// TwinCAT 3 PLC project popa_supervisor
// ProgramVersion: 3.1.4024.0
// libraries:
//   Tc2_ModbusSrv, * (Beckhoff Automation GmbH)
//   Tc2_Standard, * (Beckhoff Automation GmbH)
//   Tc2_System, * (Beckhoff Automation GmbH)
//   Tc2_Utilities, * (Beckhoff Automation GmbH)
//   Tc3_Module, * (Beckhoff Automation GmbH)
//   Tc2_OpcUa,3.3.2.0,Beckhoff Automation GmbH
// project tree:
//   DUTs/ U_Convert.TcDUT
//   GVLs/ heartbeat.TcGVL, opc.TcGVL
//   / PlcTask.TcTTO
//   POUs/ alarm_manager.TcPOU, eap_mapping.TcPOU, example_loop_control.TcPOU, faults.TcPOU, heartbeat_routine.TcPOU, interlocks.TcPOU, io_mapping.TcPOU, communications.TcPOU, general.TcPOU, modbus_mapping.TcPOU, motor_starter_control_st.TcPOU, motor_vfd_control_st.TcPOU, opc_control.TcPOU (not stored), opc_mapping.TcPOU, state_transition.TcPOU, valve_analog_control_st.TcPOU, valve_digital_control_st.TcPOU
//   POUs/Function Blocks/ int_arr_to_real.TcPOU, int_arr_to_real_1.TcPOU, modbus_analog_read.TcPOU, schneider_modbus_read.TcPOU, alarm.TcPOU, analog_scaling.TcPOU, date_time.TcPOU, motor_starter.TcPOU, motor_vfd.TcPOU, valve_analog.TcPOU, valve_digital.TcPOU
// real-time tasks:
//   TASK PlcTask: cycle T#10ms, priority 20, ADS port 350
// I/O:
//   DEVICE Device 1 (EtherCAT Automation Protocol), AmsNetId 10.60.1.100.2.1
//     Sup_Barge (Publisher)
//     Sup_Prexfer (Publisher)
//     Sup_ED (Publisher)
//     Sup_ProdXfer (Publisher)
//     Sup_Acid (Publisher)
//     Barge_Sup (Subscriber)
//     Prexfer_Sup (Subscriber)
//     ED_Sup (Subscriber)
//     ProdXfer_Sup (Subscriber)
//     Acid_Sup (Subscriber)
//   DEVICE Device 5 (EtherCAT), AmsNetId 10.60.1.100.6.1
//     Term 11 (EK1100) [EK1100 EtherCAT Coupler (2A E-Bus)]
//       Term 12 (EL2911) [EL2911, Potential supply terminal (10 A) with 4 Ch. Safety Inputs, TwinSAFE]
//         modules: Module 2 (FSOUT), Module 3 (DEVICEIO), Module 4 (FSLOGIC)
//       Term 3 (EL9011) [EL9011 End Terminal]
// variable links:
//   popa_supervisor Instance <-> Device 1 (EtherCAT Automation Protocol)/Acid_Sup (Subscriber)
//     PlcTask Inputs/eap_mapping.acid_critical_alarm <-> acid_critical_alarm/Inputs/VarData
//     PlcTask Inputs/eap_mapping.acid_error_alarm <-> acid_error_alarm/Inputs/VarData
//     PlcTask Inputs/eap_mapping.acid_warning_alarm <-> acid_warning_alarm/Inputs/VarData
//   popa_supervisor Instance <-> Device 1 (EtherCAT Automation Protocol)/Barge_Sup (Subscriber)
//     PlcTask Inputs/eap_mapping.barge_critical_alarm <-> barge_critical_alarm/Inputs/VarData
//     PlcTask Inputs/eap_mapping.barge_error_alarm <-> barge_error_alarm/Inputs/VarData
//     PlcTask Inputs/eap_mapping.barge_warning_alarm <-> barge_warning_alarm/Inputs/+
//   popa_supervisor Instance <-> Device 1 (EtherCAT Automation Protocol)/ED_Sup (Subscriber)
//     PlcTask Inputs/eap_mapping.ed_critical_alarm <-> ed_critical_alarm/Inputs/VarData
//     PlcTask Inputs/eap_mapping.ed_error_alarm <-> ed_error_alarm/Inputs/VarData
//     PlcTask Inputs/eap_mapping.ed_warning_alarm <-> ed_warning_alarm/Inputs/VarData
//   popa_supervisor Instance <-> Device 1 (EtherCAT Automation Protocol)/Prexfer_Sup (Subscriber)
//     PlcTask Inputs/eap_mapping.prexfer_critical_alarm <-> prexfer_critical_alarm/Inputs/VarData
//     PlcTask Inputs/eap_mapping.prexfer_error_alarm <-> prexfer_error_alarm/Inputs/VarData
//     PlcTask Inputs/eap_mapping.prexfer_warning_alarm <-> prexfer_warning_alarm/Inputs/VarData
//   popa_supervisor Instance <-> Device 1 (EtherCAT Automation Protocol)/ProdXfer_Sup (Subscriber)
//     PlcTask Inputs/eap_mapping.prodxfer_critical_alarm <-> prodxfer_critical_alarm/Inputs/VarData
//     PlcTask Inputs/eap_mapping.prodxfer_error_alarm <-> prodxfer_error_alarm/Inputs/VarData
//     PlcTask Inputs/eap_mapping.prodxfer_warning_alarm <-> prodxfer_warning_alarm/Inputs/VarData
//   popa_supervisor Instance <-> Device 1 (EtherCAT Automation Protocol)/Sup_Acid (Publisher)
//     PlcTask Outputs/eap_mapping.sup_acid_critical_alarm <-> sup_acid_critical_active/Outputs/VarData
//     PlcTask Outputs/eap_mapping.sup_acid_error_alarm <-> sup_acid_error_active/Outputs/VarData
//     PlcTask Outputs/eap_mapping.sup_acid_warning_alarm <-> sup_acid_warning_active/Outputs/VarData
//   popa_supervisor Instance <-> Device 1 (EtherCAT Automation Protocol)/Sup_Barge (Publisher)
//     PlcTask Outputs/eap_mapping.sup_barge_critical_alarm <-> Sup_Barge_Critical_Active/Outputs/VarData
//     PlcTask Outputs/eap_mapping.sup_barge_error_alarm <-> Sup_Barge_Error_Active/Outputs/VarData
//     PlcTask Outputs/eap_mapping.sup_barge_warning_alarm <-> Sup_Barge_Warning_Active/Outputs/VarData
//   popa_supervisor Instance <-> Device 1 (EtherCAT Automation Protocol)/Sup_ED (Publisher)
//     PlcTask Outputs/eap_mapping.sup_ed_critical_alarm <-> sup_ed_critical_active/Outputs/VarData
//     PlcTask Outputs/eap_mapping.sup_ed_error_alarm <-> sup_ed_error_active/Outputs/VarData
//     PlcTask Outputs/eap_mapping.sup_ed_warning_alarm <-> sup_ed_warning_active/Outputs/VarData
//   popa_supervisor Instance <-> Device 1 (EtherCAT Automation Protocol)/Sup_Prexfer (Publisher)
//     PlcTask Outputs/eap_mapping.sup_prexfer_critical_alarm <-> sup_prexfer_critical_active/Outputs/VarData
//     PlcTask Outputs/eap_mapping.sup_prexfer_error_alarm <-> sup_prexfer_error_active/Outputs/VarData
//     PlcTask Outputs/eap_mapping.sup_prexfer_warning_alarm <-> sup_prexfer_warning_active/Outputs/VarData
//   popa_supervisor Instance <-> Device 1 (EtherCAT Automation Protocol)/Sup_ProdXfer (Publisher)
//     PlcTask Outputs/eap_mapping.sup_prodxfer_critical_alarm <-> sup_prodxfer_critical_active/Outputs/VarData
//     PlcTask Outputs/eap_mapping.sup_prodxfer_error_alarm <-> sup_prodxfer_error_active/Outputs/VarData
//     PlcTask Outputs/eap_mapping.sup_prodxfer_warning_alarm <-> sup_prodxfer_warning_active/Outputs/VarData
//   popa_supervisor Instance <-> Device 5 (EtherCAT)/Term 11 (EK1100)/Term 12 (EL2911)
//     PlcTask Outputs/general.safety_error_ack <-> StandardOutputs/Standard In Var 1
//     PlcTask Outputs/general.safety_reset <-> StandardOutputs/Standard In Var 2
//     PlcTask Outputs/general.safety_run <-> StandardOutputs/Standard In Var 4

CONFIGURATION popa_supervisor
    RESOURCE PLC ON TwinCAT3
        TASK PlcTask(INTERVAL := T#10ms, PRIORITY := 20);
        PROGRAM communications WITH PlcTask : communications;
        PROGRAM example_loop_control WITH PlcTask : example_loop_control;
        PROGRAM faults WITH PlcTask : faults;
        PROGRAM general WITH PlcTask : general;
        PROGRAM interlocks WITH PlcTask : interlocks;
        PROGRAM io_mapping WITH PlcTask : io_mapping;
        PROGRAM opc_control WITH PlcTask : opc_control;
        PROGRAM opc_mapping WITH PlcTask : opc_mapping;
        PROGRAM state_transition WITH PlcTask : state_transition;
        PROGRAM eap_mapping WITH PlcTask : eap_mapping;
        PROGRAM alarm_manager WITH PlcTask : alarm_manager;
        PROGRAM modbus_mapping WITH PlcTask : modbus_mapping;
        PROGRAM heartbeat_routine WITH PlcTask : heartbeat_routine;
    END_RESOURCE
END_CONFIGURATION

// ---- DUTs/U_Convert.TcDUT
TYPE U_Convert :
UNION
	arrUDP_Data: ARRAY [0 .. 3] OF BYTE; // Array must start with LSB  
    rReal : REAL;
END_UNION
END_TYPE

// ---- GVLs/heartbeat.TcGVL
{attribute 'qualified_only'}
VAR_GLOBAL
	//OPC Bridge Heartbeat -- Logic found in heartbeat routine
	{attribute 'OPC.UA.DA' :='1'}
	opc_bridge_heartbeat : INT;
END_VAR

// ---- GVLs/opc.TcGVL
{attribute 'qualified_only'}
{attribute ‘OPC.UA.DA’ := ‘1’}//{attribute 'global_init_slot' := '50500'}
VAR_GLOBAL PERSISTENT
	//These tags are created here because you cannot write directly to local scoped tags(cpt_3144) from outside the POU
	//They are created here then mapped to the local variables in the POU
	//All tags in this GVL MUST have the {attribute 'OPC.UA.DA' :='1'} string above them in order to be exposed to OPC
	//Tags that are ONLY being read from the HMI have their values set in the opc_mapping program
		
	
	//--- Heartbeat ------------------------------------------------------------------------------------------------
	{attribute 'OPC.UA.DA' :='1'}
	popa_supervisor_opc_bridge_heartbeat : BOOL;
	
	//--- Safety ---------------------------------------------------------------------------------------------------
	{attribute 'OPC.UA.DA' :='1'}
	popa_supervisor_safety_reset : BOOL;
	
	{attribute 'OPC.UA.DA' :='1'}
	popa_supervisor_estop_active : BOOL;
	
	{attribute 'OPC.UA.DA' :='1'}
	popa_supervisor_barge_safety_triggered : BOOL;

	{attribute 'OPC.UA.DA' :='1'}
	popa_supervisor_ptt_safety_triggered : BOOL;

	{attribute 'OPC.UA.DA' :='1'}
	popa_supervisor_ed_safety_triggered : BOOL;

	{attribute 'OPC.UA.DA' :='1'}
	popa_supervisor_pdt_safety_triggered : BOOL;

	{attribute 'OPC.UA.DA' :='1'}
	popa_supervisor_acid_safety_triggered : BOOL;


	//--- Macoma Power Meters --------------------------------------------------------------------------------------

	{attribute 'OPC.UA.DA' :='1'}
	popa_supervisor_kt_3710_line_to_neutral_voltage_scaled_value : REAL;
	{attribute 'OPC.UA.DA' :='1'}
	popa_supervisor_kt_3710_line_to_line_voltage_scaled_value : REAL;
	{attribute 'OPC.UA.DA' :='1'}
	popa_supervisor_kt_3710_avg_line_current_scaled_value : REAL;
	{attribute 'OPC.UA.DA' :='1'}
	popa_supervisor_kt_3710_total_active_power_scaled_value : REAL;
	{attribute 'OPC.UA.DA' :='1'}
	popa_supervisor_kt_3710_total_reactive_power_scaled_value : REAL;
	{attribute 'OPC.UA.DA' :='1'}
	popa_supervisor_kt_3710_total_apparent_power_scaled_value : REAL;
	{attribute 'OPC.UA.DA' :='1'}
	popa_supervisor_kt_3710_total_power_factor_scaled_value : REAL;
	{attribute 'OPC.UA.DA' :='1'}
	popa_supervisor_kt_3710_system_frequency_scaled_value : REAL;
	
	{attribute 'OPC.UA.DA' :='1'}
	popa_supervisor_kt_3715_line_to_neutral_voltage_scaled_value : REAL;
	{attribute 'OPC.UA.DA' :='1'}
	popa_supervisor_kt_3715_line_to_line_voltage_scaled_value : REAL;
	{attribute 'OPC.UA.DA' :='1'}
	popa_supervisor_kt_3715_avg_line_current_scaled_value : REAL;
	{attribute 'OPC.UA.DA' :='1'}
	popa_supervisor_kt_3715_total_active_power_scaled_value : REAL;
	{attribute 'OPC.UA.DA' :='1'}
	popa_supervisor_kt_3715_total_reactive_power_scaled_value : REAL;
	{attribute 'OPC.UA.DA' :='1'}
	popa_supervisor_kt_3715_total_apparent_power_scaled_value : REAL;
	{attribute 'OPC.UA.DA' :='1'}
	popa_supervisor_kt_3715_total_power_factor_scaled_value : REAL;
	{attribute 'OPC.UA.DA' :='1'}
	popa_supervisor_kt_3715_system_frequency_scaled_value : REAL;
	
	{attribute 'OPC.UA.DA' :='1'}
	popa_supervisor_kt_2710_line_to_neutral_voltage_scaled_value : REAL;
	{attribute 'OPC.UA.DA' :='1'}
	popa_supervisor_kt_2710_line_to_line_voltage_scaled_value : REAL;
	{attribute 'OPC.UA.DA' :='1'}
	popa_supervisor_kt_2710_avg_line_current_scaled_value : REAL;
	{attribute 'OPC.UA.DA' :='1'}
	popa_supervisor_kt_2710_total_active_power_scaled_value : REAL;
	{attribute 'OPC.UA.DA' :='1'}
	popa_supervisor_kt_2710_total_reactive_power_scaled_value : REAL;
	{attribute 'OPC.UA.DA' :='1'}
	popa_supervisor_kt_2710_total_apparent_power_scaled_value : REAL;
	{attribute 'OPC.UA.DA' :='1'}
	popa_supervisor_kt_2710_total_power_factor_scaled_value : REAL;
	{attribute 'OPC.UA.DA' :='1'}
	popa_supervisor_kt_2710_system_frequency_scaled_value : REAL;
	
	{attribute 'OPC.UA.DA' :='1'}
	popa_supervisor_kt_2715_line_to_neutral_voltage_scaled_value : REAL;
	{attribute 'OPC.UA.DA' :='1'}
	popa_supervisor_kt_2715_line_to_line_voltage_scaled_value : REAL;
	{attribute 'OPC.UA.DA' :='1'}
	popa_supervisor_kt_2715_avg_line_current_scaled_value : REAL;
	{attribute 'OPC.UA.DA' :='1'}
	popa_supervisor_kt_2715_total_active_power_scaled_value : REAL;
	{attribute 'OPC.UA.DA' :='1'}
	popa_supervisor_kt_2715_total_reactive_power_scaled_value : REAL;
	{attribute 'OPC.UA.DA' :='1'}
	popa_supervisor_kt_2715_total_apparent_power_scaled_value : REAL;
	{attribute 'OPC.UA.DA' :='1'}
	popa_supervisor_kt_2715_total_power_factor_scaled_value : REAL;
	{attribute 'OPC.UA.DA' :='1'}
	popa_supervisor_kt_2715_system_frequency_scaled_value : REAL;
	
	
	{attribute 'OPC.UA.DA' :='1'}
	popa_supervisor_kt_2720_line_to_neutral_voltage_scaled_value : REAL;
	{attribute 'OPC.UA.DA' :='1'}
	popa_supervisor_kt_2720_line_to_line_voltage_scaled_value : REAL;
	{attribute 'OPC.UA.DA' :='1'}
	popa_supervisor_kt_2720_avg_line_current_scaled_value : REAL;
	{attribute 'OPC.UA.DA' :='1'}
	popa_supervisor_kt_2720_total_active_power_scaled_value : REAL;
	{attribute 'OPC.UA.DA' :='1'}
	popa_supervisor_kt_2720_total_reactive_power_scaled_value : REAL;
	{attribute 'OPC.UA.DA' :='1'}
	popa_supervisor_kt_2720_total_apparent_power_scaled_value : REAL;
	{attribute 'OPC.UA.DA' :='1'}
	popa_supervisor_kt_2720_total_power_factor_scaled_value : REAL;
	{attribute 'OPC.UA.DA' :='1'}
	popa_supervisor_kt_2720_system_frequency_scaled_value : REAL;
	
	{attribute 'OPC.UA.DA' :='1'}
	popa_supervisor_kt_2725_line_to_neutral_voltage_scaled_value : REAL;
	{attribute 'OPC.UA.DA' :='1'}
	popa_supervisor_kt_2725_line_to_line_voltage_scaled_value : REAL;
	{attribute 'OPC.UA.DA' :='1'}
	popa_supervisor_kt_2725_avg_line_current_scaled_value : REAL;
	{attribute 'OPC.UA.DA' :='1'}
	popa_supervisor_kt_2725_total_active_power_scaled_value : REAL;
	{attribute 'OPC.UA.DA' :='1'}
	popa_supervisor_kt_2725_total_reactive_power_scaled_value : REAL;
	{attribute 'OPC.UA.DA' :='1'}
	popa_supervisor_kt_2725_total_apparent_power_scaled_value : REAL;
	{attribute 'OPC.UA.DA' :='1'}
	popa_supervisor_kt_2725_total_power_factor_scaled_value : REAL;
	{attribute 'OPC.UA.DA' :='1'}
	popa_supervisor_kt_2725_system_frequency_scaled_value : REAL;
	
	{attribute 'OPC.UA.DA' :='1'}
	popa_supervisor_kt_2730_line_to_neutral_voltage_scaled_value : REAL;
	{attribute 'OPC.UA.DA' :='1'}
	popa_supervisor_kt_2730_line_to_line_voltage_scaled_value : REAL;
	{attribute 'OPC.UA.DA' :='1'}
	popa_supervisor_kt_2730_avg_line_current_scaled_value : REAL;
	{attribute 'OPC.UA.DA' :='1'}
	popa_supervisor_kt_2730_total_active_power_scaled_value : REAL;
	{attribute 'OPC.UA.DA' :='1'}
	popa_supervisor_kt_2730_total_reactive_power_scaled_value : REAL;
	{attribute 'OPC.UA.DA' :='1'}
	popa_supervisor_kt_2730_total_apparent_power_scaled_value : REAL;
	{attribute 'OPC.UA.DA' :='1'}
	popa_supervisor_kt_2730_total_power_factor_scaled_value : REAL;
	{attribute 'OPC.UA.DA' :='1'}
	popa_supervisor_kt_2730_system_frequency_scaled_value : REAL;
	
	{attribute 'OPC.UA.DA' :='1'}
	popa_supervisor_kt_3720_line_to_neutral_voltage_scaled_value : REAL;
	{attribute 'OPC.UA.DA' :='1'}
	popa_supervisor_kt_3720_line_to_line_voltage_scaled_value : REAL;
	{attribute 'OPC.UA.DA' :='1'}
	popa_supervisor_kt_3720_avg_line_current_scaled_value : REAL;
	{attribute 'OPC.UA.DA' :='1'}
	popa_supervisor_kt_3720_total_active_power_scaled_value : REAL;
	{attribute 'OPC.UA.DA' :='1'}
	popa_supervisor_kt_3720_total_reactive_power_scaled_value : REAL;
	{attribute 'OPC.UA.DA' :='1'}
	popa_supervisor_kt_3720_total_apparent_power_scaled_value : REAL;
	{attribute 'OPC.UA.DA' :='1'}
	popa_supervisor_kt_3720_total_power_factor_scaled_value : REAL;
	{attribute 'OPC.UA.DA' :='1'}
	popa_supervisor_kt_3720_system_frequency_scaled_value : REAL;
	
	{attribute 'OPC.UA.DA' :='1'}
	popa_supervisor_kt_1720_line_to_neutral_voltage_scaled_value : REAL;
	{attribute 'OPC.UA.DA' :='1'}
	popa_supervisor_kt_1720_line_to_line_voltage_scaled_value : REAL;
	{attribute 'OPC.UA.DA' :='1'}
	popa_supervisor_kt_1720_avg_line_current_scaled_value : REAL;
	{attribute 'OPC.UA.DA' :='1'}
	popa_supervisor_kt_1720_total_active_power_scaled_value : REAL;
	{attribute 'OPC.UA.DA' :='1'}
	popa_supervisor_kt_1720_total_reactive_power_scaled_value : REAL;
	{attribute 'OPC.UA.DA' :='1'}
	popa_supervisor_kt_1720_total_apparent_power_scaled_value : REAL;
	{attribute 'OPC.UA.DA' :='1'}
	popa_supervisor_kt_1720_total_power_factor_scaled_value : REAL;
	{attribute 'OPC.UA.DA' :='1'}
	popa_supervisor_kt_1720_system_frequency_scaled_value : REAL;
	
	{attribute 'OPC.UA.DA' :='1'}
	popa_supervisor_kt_4710_line_to_neutral_voltage_scaled_value : REAL;
	{attribute 'OPC.UA.DA' :='1'}
	popa_supervisor_kt_4710_line_to_line_voltage_scaled_value : REAL;
	{attribute 'OPC.UA.DA' :='1'}
	popa_supervisor_kt_4710_avg_line_current_scaled_value : REAL;
	{attribute 'OPC.UA.DA' :='1'}
	popa_supervisor_kt_4710_total_active_power_scaled_value : REAL;
	{attribute 'OPC.UA.DA' :='1'}
	popa_supervisor_kt_4710_total_reactive_power_scaled_value : REAL;
	{attribute 'OPC.UA.DA' :='1'}
	popa_supervisor_kt_4710_total_apparent_power_scaled_value : REAL;
	{attribute 'OPC.UA.DA' :='1'}
	popa_supervisor_kt_4710_total_power_factor_scaled_value : REAL;
	{attribute 'OPC.UA.DA' :='1'}
	popa_supervisor_kt_4710_system_frequency_scaled_value : REAL;
	
	{attribute 'OPC.UA.DA' :='1'}
	popa_supervisor_kt_1725_line_to_neutral_voltage_scaled_value : REAL;
	{attribute 'OPC.UA.DA' :='1'}
	popa_supervisor_kt_1725_line_to_line_voltage_scaled_value : REAL;
	{attribute 'OPC.UA.DA' :='1'}
	popa_supervisor_kt_1725_avg_line_current_scaled_value : REAL;
	{attribute 'OPC.UA.DA' :='1'}
	popa_supervisor_kt_1725_total_active_power_scaled_value : REAL;
	{attribute 'OPC.UA.DA' :='1'}
	popa_supervisor_kt_1725_total_reactive_power_scaled_value : REAL;
	{attribute 'OPC.UA.DA' :='1'}
	popa_supervisor_kt_1725_total_apparent_power_scaled_value : REAL;
	{attribute 'OPC.UA.DA' :='1'}
	popa_supervisor_kt_1725_total_power_factor_scaled_value : REAL;
	{attribute 'OPC.UA.DA' :='1'}
	popa_supervisor_kt_1725_system_frequency_scaled_value : REAL;
	
	{attribute 'OPC.UA.DA' :='1'}
	popa_supervisor_kt_1715_line_to_neutral_voltage_scaled_value : REAL;
	{attribute 'OPC.UA.DA' :='1'}
	popa_supervisor_kt_1715_line_to_line_voltage_scaled_value : REAL;
	{attribute 'OPC.UA.DA' :='1'}
	popa_supervisor_kt_1715_avg_line_current_scaled_value : REAL;
	{attribute 'OPC.UA.DA' :='1'}
	popa_supervisor_kt_1715_total_active_power_scaled_value : REAL;
	{attribute 'OPC.UA.DA' :='1'}
	popa_supervisor_kt_1715_total_reactive_power_scaled_value : REAL;
	{attribute 'OPC.UA.DA' :='1'}
	popa_supervisor_kt_1715_total_apparent_power_scaled_value : REAL;
	{attribute 'OPC.UA.DA' :='1'}
	popa_supervisor_kt_1715_total_power_factor_scaled_value : REAL;
	{attribute 'OPC.UA.DA' :='1'}
	popa_supervisor_kt_1715_system_frequency_scaled_value : REAL;
	{attribute 'OPC.UA.DA' :='1'}
	popa_supervisor_kt_1715_ground_current_scaled_value : REAL;
	{attribute 'OPC.UA.DA' :='1'}
	popa_supervisor_kt_1715_current_capacity_scaled_value : REAL;
	{attribute 'OPC.UA.DA' :='1'}
	popa_supervisor_kt_1715_power_factor_leading_scaled_value : REAL;
	{attribute 'OPC.UA.DA' :='1'}
	popa_supervisor_kt_1715_power_factor_lagging_scaled_value : REAL;
	
	{attribute 'OPC.UA.DA' :='1'}
	popa_supervisor_kt_1710_line_to_neutral_voltage_scaled_value : REAL;
	{attribute 'OPC.UA.DA' :='1'}
	popa_supervisor_kt_1710_line_to_line_voltage_scaled_value : REAL;
	{attribute 'OPC.UA.DA' :='1'}
	popa_supervisor_kt_1710_avg_line_current_scaled_value : REAL;
	{attribute 'OPC.UA.DA' :='1'}
	popa_supervisor_kt_1710_total_active_power_scaled_value : REAL;
	{attribute 'OPC.UA.DA' :='1'}
	popa_supervisor_kt_1710_total_reactive_power_scaled_value : REAL;
	{attribute 'OPC.UA.DA' :='1'}
	popa_supervisor_kt_1710_total_apparent_power_scaled_value : REAL;
	{attribute 'OPC.UA.DA' :='1'}
	popa_supervisor_kt_1710_total_power_factor_scaled_value : REAL;
	{attribute 'OPC.UA.DA' :='1'}
	popa_supervisor_kt_1710_system_frequency_scaled_value : REAL;
	{attribute 'OPC.UA.DA' :='1'}
	popa_supervisor_kt_1710_ground_current_scaled_value : REAL;
	{attribute 'OPC.UA.DA' :='1'}
	popa_supervisor_kt_1710_current_capacity_scaled_value : REAL;
	{attribute 'OPC.UA.DA' :='1'}
	popa_supervisor_kt_1710_power_factor_leading_scaled_value : REAL;
	{attribute 'OPC.UA.DA' :='1'}
	popa_supervisor_kt_1710_power_factor_lagging_scaled_value : REAL;

END_VAR

// ---- POUs/communications.TcPOU
PROGRAM communications
VAR PERSISTENT
END_VAR

END_PROGRAM

// ---- POUs/example_loop_control.TcPOU
PROGRAM example_loop_control
VAR

END_VAR

// NETWORK 1

END_PROGRAM

// ---- POUs/faults.TcPOU
PROGRAM faults
VAR PERSISTENT
	// Example analog alarm low low
	cpt_3144_low_low: Alarm;
	// Example analog alarm low
	cpt_3144_low: Alarm;
	// Example analog alarm high
	cpt_3144_high: Alarm;
	// Example analog alarm high high
	cpt_3144_high_high: Alarm;
END_VAR

(*//Instantiate the alarm block, and map the inputs from the OPC GVL
cpt_3144_low_low();
cpt_3144_low_low.alm_ack:=opc.popa_0081_alarm_ack;
cpt_3144_low_low.reset:=opc.popa_0081_alarm_reset;
cpt_3144_low_low.priority:=opc.popa_0081_cpt_3144_low_low_priority;
cpt_3144_low_low.delay_setpoint:=opc.popa_0081_cpt_3144_low_low_delay_setpoint;
cpt_3144_low_low.enable:=opc.popa_0081_cpt_3144_low_low_enable;

//Place your alarm trigger logic here.  
IF io_mapping.cpt_3144.scaled_value<opc.popa_0081_cpt_3144_low_low_setpoint THEN
	cpt_3144_low_low.trigger:=TRUE;
	ELSE
		cpt_3144_low_low.trigger:=FALSE;
	END_IF	
	
//Instantiate the alarm block, and map the inputs from the OPC GVL
cpt_3144_low();
cpt_3144_low.alm_ack:=opc.popa_0081_alarm_ack;
cpt_3144_low.reset:=opc.popa_0081_alarm_reset;
cpt_3144_low.priority:=opc.popa_0081_cpt_3144_low_priority;
cpt_3144_low.delay_setpoint:=opc.popa_0081_cpt_3144_low_delay_setpoint;
cpt_3144_low.enable:=opc.popa_0081_cpt_3144_low_enable;

//Place your alarm trigger logic here.  
IF io_mapping.cpt_3144.scaled_value<opc.popa_0081_cpt_3144_low_setpoint THEN
	cpt_3144_low.trigger:=TRUE;
	ELSE
		cpt_3144_low.trigger:=FALSE;
	END_IF
	
//Instantiate the alarm block, and map the inputs from the OPC GVL
cpt_3144_high();
cpt_3144_high.alm_ack:=opc.popa_0081_alarm_ack;
cpt_3144_high.reset:=opc.popa_0081_alarm_reset;
cpt_3144_high.priority:=opc.popa_0081_cpt_3144_high_priority;
cpt_3144_high.delay_setpoint:=opc.popa_0081_cpt_3144_high_delay_setpoint;
cpt_3144_high.enable:=opc.popa_0081_cpt_3144_high_enable;

//Place your alarm trigger logic here.  
IF io_mapping.cpt_3144.scaled_value<opc.popa_0081_cpt_3144_high_setpoint THEN
	cpt_3144_high.trigger:=TRUE;
	ELSE
		cpt_3144_high.trigger:=FALSE;
	END_IF
	
//Instantiate the alarm block, and map the inputs from the OPC GVL
cpt_3144_high_high();
cpt_3144_high_high.alm_ack:=opc.popa_0081_alarm_ack;
cpt_3144_high_high.reset:=opc.popa_0081_alarm_reset;
cpt_3144_high_high.priority:=opc.popa_0081_cpt_3144_high_high_priority;
cpt_3144_high_high.delay_setpoint:=opc.popa_0081_cpt_3144_high_high_delay_setpoint;
cpt_3144_high_high.enable:=opc.popa_0081_cpt_3144_high_high_enable;

//Place your alarm trigger logic here.  
IF io_mapping.cpt_3144.scaled_value<opc.popa_0081_cpt_3144_high_high_setpoint THEN
	cpt_3144_high_high.trigger:=TRUE;
	ELSE
		cpt_3144_high_high.trigger:=FALSE;
	END_IF
	*)

END_PROGRAM

// ---- POUs/Function Blocks/alarm.TcPOU
FUNCTION_BLOCK alarm
VAR_INPUT
	//Input that triggers the alarm condition
	trigger : BOOL;
	//Alarm Acknowledge bit, Clears low priority alarms
	alm_ack : BOOL;
	//Alarm Reset, clears high priority alarms
	reset : BOOL;
	//Alarm Priority, 1=Warning, 2=Error, 3=Critical
	priority : INT;
	//Alarm Delay Setpoint in Seconds
	delay_setpoint : INT;
	//Alarm Enable
	enable : BOOL;
END_VAR
VAR_OUTPUT
	//Alarm is triggered
	active : BOOL;
END_VAR
VAR
	//Delay Timer Tags
	delay_ton : TON;
	delay_ton_pt : TIME;
	delay_ton_et : TIME;
	//Delay setpoint converted to Milliseconds
	delay_ms : REAL;
	//Cutoff for needing to reset vs ack an alarm.  At or above this value requires reset.  
	reset_priority : REAL :=3;
END_VAR

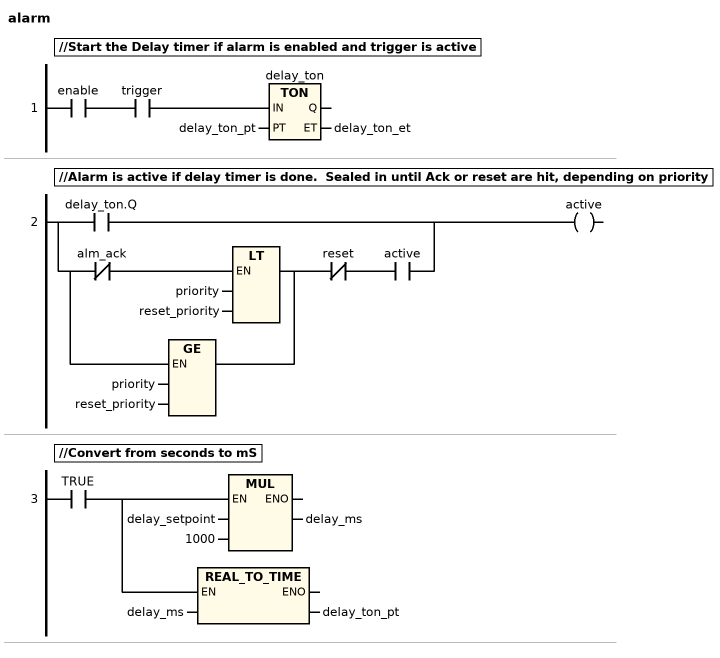
// NETWORK 1
// label: //Start the Delay timer if alarm is enabled and trigger is active
delay_ton(IN := enable AND trigger, PT := delay_ton_pt, ET => delay_ton_et); // TON

// NETWORK 2
// label: //Alarm is active if delay timer is done.  Sealed in until Ack or reset are hit, depending on priority
active := delay_ton.Q OR (NOT alm_ack AND priority < reset_priority OR priority >= reset_priority) AND NOT reset AND active;

// NETWORK 3
// label: //Convert from seconds to mS
delay_ms := delay_setpoint * 1000;
delay_ton_pt := REAL_TO_TIME(delay_ms);

END_FUNCTION_BLOCK

// ---- POUs/general.TcPOU
PROGRAM general
VAR PERSISTENT
	//System date time function block
	system_date_time : date_time;
	//Daily reset bit, used throughout the program for any resets
	daily_reset : BOOL;
	//Alarm Acknoweldge unlatch timer
	alarm_ack_ton : ton;
	//Alarm Reset unlatch timer
	alarm_reset_ton : ton;
	//Alarm Ack and reset unlatch timer setpoint
	alarm_ack_unlatch_sp : TIME :=T#3S;
	
	safety_reset_ton : TON;
	
	safety_reset AT %Q*  : BOOL;
	safety_error_ack AT %Q* : BOOL;
	safety_run AT %Q*  : BOOL;
	
END_VAR

VAR
	
	safety_reset_ons: R_TRIG;
END_VAR
VAR // added by the converter: edge detectors and wires of the graphical bodies
    _w1 : BOOL;
END_VAR

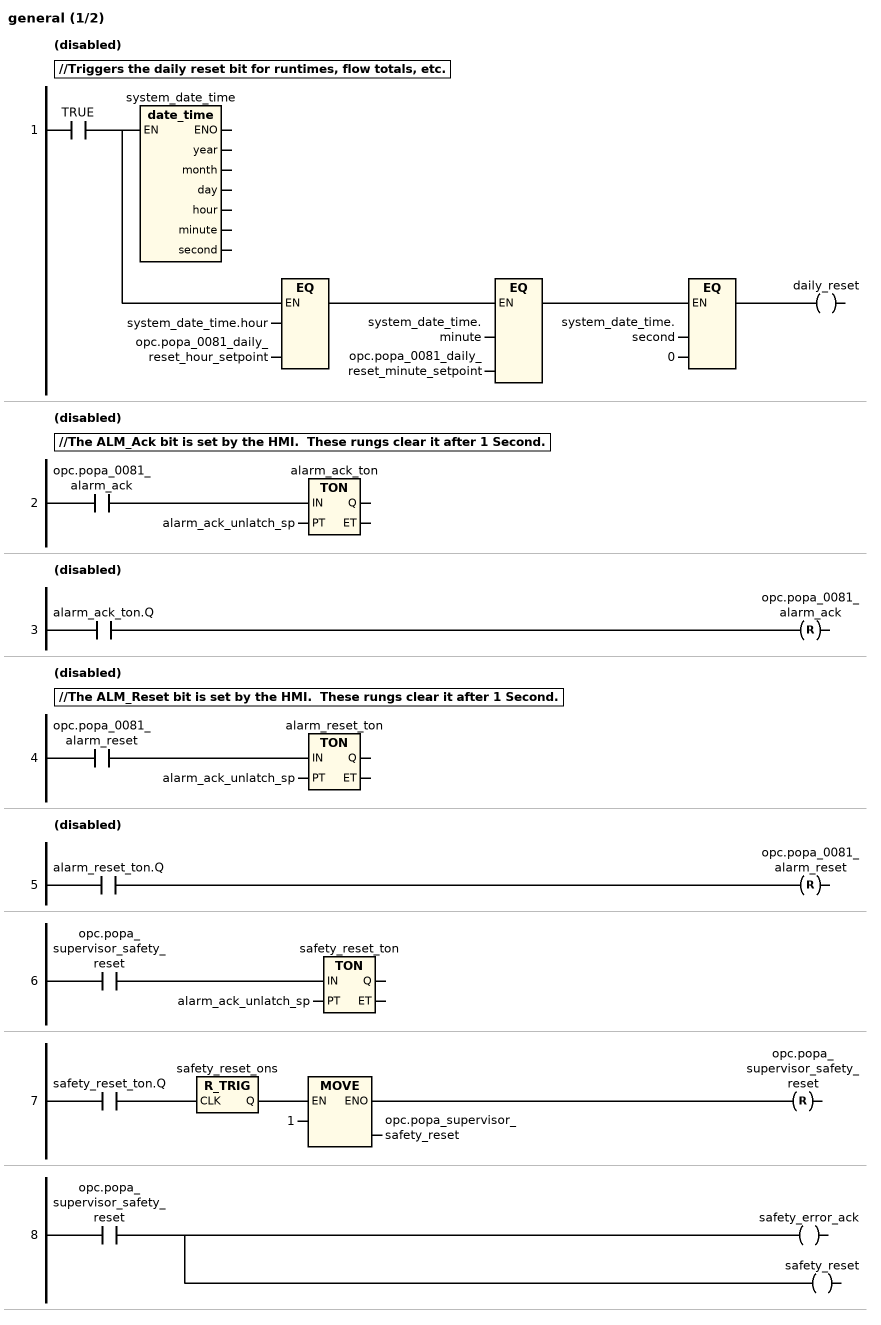
// NETWORK 1 (disabled)
// label: //Triggers the daily reset bit for runtimes, flow totals, etc.
// system_date_time(); // date_time
// daily_reset := system_date_time.hour = opc.popa_0081_daily_reset_hour_setpoint AND system_date_time.minute = opc.popa_0081_daily_reset_minute_setpoint AND system_date_time.second = 0;

// NETWORK 2 (disabled)
// label: //The ALM_Ack bit is set by the HMI.  These rungs clear it after 1 Second.
// alarm_ack_ton(IN := opc.popa_0081_alarm_ack, PT := alarm_ack_unlatch_sp); // TON

// NETWORK 3 (disabled)
// opc.popa_0081_alarm_ack R= alarm_ack_ton.Q;

// NETWORK 4 (disabled)
// label: //The ALM_Reset bit is set by the HMI.  These rungs clear it after 1 Second.
// alarm_reset_ton(IN := opc.popa_0081_alarm_reset, PT := alarm_ack_unlatch_sp); // TON

// NETWORK 5 (disabled)
// opc.popa_0081_alarm_reset R= alarm_reset_ton.Q;

// NETWORK 6
safety_reset_ton(IN := opc.popa_supervisor_safety_reset, PT := alarm_ack_unlatch_sp); // TON

// NETWORK 7
safety_reset_ons(CLK := safety_reset_ton.Q); // R_TRIG
_w1 := safety_reset_ons.Q;
IF _w1 THEN opc.popa_supervisor_safety_reset := 1; END_IF
opc.popa_supervisor_safety_reset R= _w1;

// NETWORK 8
safety_error_ack := opc.popa_supervisor_safety_reset;
safety_reset := opc.popa_supervisor_safety_reset;

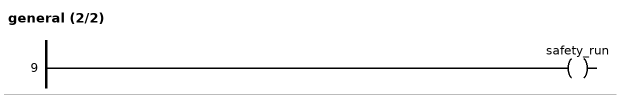
// NETWORK 9
safety_run := TRUE;

END_PROGRAM

// ---- POUs/Function Blocks/date_time.TcPOU
FUNCTION_BLOCK Date_Time
VAR_INPUT
END_VAR
VAR_OUTPUT
	Year : INT;
	Month : INT;
	Day : INT;
	Hour : INT;
	Minute : INT;
	Second : INT;
END_VAR
VAR
	fbGetSystemTime : GETSYSTEMTIME;    (*timestamp*)
    fileTime        : T_FILETIME;
    sDT: STRING(30);
END_VAR

//Get Timestamp from System
fbGetSystemTime(timeLoDW => fileTime.dwLowDateTime, timeHiDW => fileTime.dwHighDateTime);
//Convert from systemtime to string, this makes it easier to break out into Ints for Logic usage.
sDT := SYSTEMTIME_TO_STRING(FILETIME_TO_SYSTEMTIME(fileTime));
//Breakout string into individual Ints.
Year := STRING_TO_INT(LEFT(sDt, 4));
Month := STRING_TO_INT(MID(sDt, 2, 6));
Day := STRING_TO_INT(MID(sDt, 2, 9));
Hour := STRING_TO_INT(MID(sDt, 2, 12));
Minute := STRING_TO_INT(MID(sDt, 2, 15));
Second := STRING_TO_INT(MID(sDt, 2, 18));

END_FUNCTION_BLOCK

// ---- POUs/interlocks.TcPOU
PROGRAM interlocks
VAR PERSISTENT
END_VAR

// NETWORK 1

END_PROGRAM

// ---- POUs/io_mapping.TcPOU
PROGRAM io_mapping
VAR PERSISTENT
    //Example analog input function block
    cpt_3144 : analog_scaling;
	
	test_real AT %Q* : REAL;
	
	publisharray AT %Q* : ARRAY[0..9] OF REAL;
	
	sine_wave : REAL;
	
    //Example Analog input raw input, mapped to a physical input
    cpt_3144_raw_input AT %I* : INT;

END_VAR

(*//Instantiate Example analog input function block
cpt_3144();

//Map values from the OPC GVL so that they can be written to from outside POU(IE from HMI)
cpt_3144.eu_max:=opc.popa_0081_cpt_3144_eu_max;
cpt_3144.eu_min:=opc.popa_0081_cpt_3144_eu_min;
cpt_3144.filter_factor:=opc.popa_0081_cpt_3144_filter_factor;
cpt_3144.raw_max:=opc.popa_0081_cpt_3144_raw_max;
cpt_3144.raw_min:=opc.popa_0081_cpt_3144_raw_min;
//Map the analog scaling function block raw input to the physical raw input variable
cpt_3144.raw_input := cpt_3144_raw_input;

sine_wave:=sine_wave+0.001;
IF (sine_wave>(2*pi)) THEN
	sine_wave:=0;
END_IF
*)
publisharray[0]:=sine_wave;
publisharray[1]:=sine_wave/2;
publisharray[2]:=sine_wave*2;

END_PROGRAM

// ---- POUs/Function Blocks/analog_scaling.TcPOU
FUNCTION_BLOCK Analog_Scaling
VAR_INPUT
	//Raw Input value
	Raw_Input : REAL;
	//Raw Input Minimum Scaling Value
	Raw_Min : REAL;
	//Raw Input Maximum Scaling Value
	Raw_Max : REAL;
	//Engineering Units Minimum Scaling Value
	EU_Min : REAL;
	//Engineering Units Maximum Scaling Value
	EU_Max : REAL;
	//Averaging Filter Time Setpoint
	Filter_Factor : REAL;
END_VAR
VAR_OUTPUT
	//Scaled Value for Output
	Scaled_Value : REAL;
END_VAR
VAR
	//Scratchpad Value
	Normalized_Value : REAL;
	//Normalized/Scaled Value
	Scaled : REAL;
END_VAR

//Initialize Raw_Max and EU_Max to avoid Scaled_Value=Not a number
IF Raw_Max = 0 AND Raw_Min = 0 THEN
	Raw_Max:=1;
END_IF
IF EU_Max = 0 AND Raw_Min = 0 THEN
	EU_Max:=1;
END_IF

//Normalize the Analog Input
IF Raw_Input < Raw_Min THEN
		Normalized_Value := Raw_Min;
	ELSIF Raw_Input > Raw_Max THEN
		Normalized_Value := Raw_Max;
	ELSE
		Normalized_Value := (Raw_Input - Raw_Min) / (Raw_Max - Raw_Min);
	END_IF
	
//Scale the Output
Scaled := Normalized_Value * (EU_Max-EU_Min)+EU_Min;

//Low Pass Filter for the output.  Increase Filter to dampen reading
Scaled_Value := ((Scaled_Value * Filter_Factor) + Scaled) / (Filter_Factor +1);

END_FUNCTION_BLOCK

// ---- POUs/opc_mapping.TcPOU
PROGRAM opc_mapping
VAR
END_VAR

//This program maps values from the local variable to the OPC readable tag.
// --- Hearbeat ------------------------------------------------------------------------------------------------------------------------------------
opc.popa_supervisor_opc_bridge_heartbeat := NOT(heartbeat_routine.opc_heartbeat_error);

// --- Safety Logging ------------------------------------------------------------------------------------------------------------------------------
opc.popa_supervisor_barge_safety_triggered := eap_mapping.barge_critical_alarm;
opc.popa_supervisor_ptt_safety_triggered := eap_mapping.prexfer_critical_alarm;
opc.popa_supervisor_ed_safety_triggered := eap_mapping.ed_critical_alarm;
opc.popa_supervisor_pdt_safety_triggered := eap_mapping.prodxfer_critical_alarm;
opc.popa_supervisor_acid_safety_triggered := eap_mapping.acid_critical_alarm;

// --- Power Meter Data ----------------------------------------------------------------------------------------------------------------------------
opc.popa_supervisor_kt_3710_line_to_neutral_voltage_scaled_value := modbus_mapping.bped_main_power_meter_modbus_read.avg_line_to_neutral_voltage;

opc.popa_supervisor_kt_3710_line_to_line_voltage_scaled_value := modbus_mapping.bped_main_power_meter_modbus_read.avg_line_to_line_voltage;

opc.popa_supervisor_kt_3710_avg_line_current_scaled_value := modbus_mapping.bped_main_power_meter_modbus_read.system_avg_line_current;

opc.popa_supervisor_kt_3710_total_active_power_scaled_value := modbus_mapping.bped_main_power_meter_modbus_read.total_active_power;

opc.popa_supervisor_kt_3710_total_reactive_power_scaled_value := modbus_mapping.bped_main_power_meter_modbus_read.total_reactive_power;

opc.popa_supervisor_kt_3710_total_apparent_power_scaled_value := modbus_mapping.bped_main_power_meter_modbus_read.total_apparent_power;

opc.popa_supervisor_kt_3710_total_power_factor_scaled_value := modbus_mapping.bped_main_power_meter_modbus_read.total_power_factor;

opc.popa_supervisor_kt_3710_system_frequency_scaled_value := modbus_mapping.bped_main_power_meter_modbus_read.system_frequency;

opc.popa_supervisor_kt_3715_line_to_neutral_voltage_scaled_value := modbus_mapping.bped_stack_power_meter_modbus_read.avg_line_to_neutral_voltage;

opc.popa_supervisor_kt_3715_line_to_line_voltage_scaled_value := modbus_mapping.bped_stack_power_meter_modbus_read.avg_line_to_line_voltage;

opc.popa_supervisor_kt_3715_avg_line_current_scaled_value := modbus_mapping.bped_stack_power_meter_modbus_read.system_avg_line_current;

opc.popa_supervisor_kt_3715_total_active_power_scaled_value := modbus_mapping.bped_stack_power_meter_modbus_read.total_active_power;

opc.popa_supervisor_kt_3715_total_reactive_power_scaled_value := modbus_mapping.bped_stack_power_meter_modbus_read.total_reactive_power;

opc.popa_supervisor_kt_3715_total_apparent_power_scaled_value := modbus_mapping.bped_stack_power_meter_modbus_read.total_apparent_power;

opc.popa_supervisor_kt_3715_total_power_factor_scaled_value := modbus_mapping.bped_stack_power_meter_modbus_read.total_power_factor;

opc.popa_supervisor_kt_3715_system_frequency_scaled_value := modbus_mapping.bped_stack_power_meter_modbus_read.system_frequency;


opc.popa_supervisor_kt_2710_line_to_neutral_voltage_scaled_value := modbus_mapping.nf1_power_meter_modbus_read.avg_line_to_neutral_voltage;

opc.popa_supervisor_kt_2710_line_to_line_voltage_scaled_value := modbus_mapping.nf1_power_meter_modbus_read.avg_line_to_line_voltage;

opc.popa_supervisor_kt_2710_avg_line_current_scaled_value := modbus_mapping.nf1_power_meter_modbus_read.system_avg_line_current;

opc.popa_supervisor_kt_2710_total_active_power_scaled_value := modbus_mapping.nf1_power_meter_modbus_read.total_active_power;

opc.popa_supervisor_kt_2710_total_reactive_power_scaled_value := modbus_mapping.nf1_power_meter_modbus_read.total_reactive_power;

opc.popa_supervisor_kt_2710_total_apparent_power_scaled_value := modbus_mapping.nf1_power_meter_modbus_read.total_apparent_power;

opc.popa_supervisor_kt_2710_total_power_factor_scaled_value := modbus_mapping.nf1_power_meter_modbus_read.total_power_factor;

opc.popa_supervisor_kt_2710_system_frequency_scaled_value := modbus_mapping.nf1_power_meter_modbus_read.system_frequency;


opc.popa_supervisor_kt_2715_line_to_neutral_voltage_scaled_value := modbus_mapping.nf2_power_meter_modbus_read.avg_line_to_neutral_voltage;

opc.popa_supervisor_kt_2715_line_to_line_voltage_scaled_value := modbus_mapping.nf2_power_meter_modbus_read.avg_line_to_line_voltage;

opc.popa_supervisor_kt_2715_avg_line_current_scaled_value := modbus_mapping.nf2_power_meter_modbus_read.system_avg_line_current;

opc.popa_supervisor_kt_2715_total_active_power_scaled_value := modbus_mapping.nf2_power_meter_modbus_read.total_active_power;

opc.popa_supervisor_kt_2715_total_reactive_power_scaled_value := modbus_mapping.nf2_power_meter_modbus_read.total_reactive_power;

opc.popa_supervisor_kt_2715_total_apparent_power_scaled_value := modbus_mapping.nf2_power_meter_modbus_read.total_apparent_power;

opc.popa_supervisor_kt_2715_total_power_factor_scaled_value := modbus_mapping.nf2_power_meter_modbus_read.total_power_factor;

opc.popa_supervisor_kt_2715_system_frequency_scaled_value := modbus_mapping.nf2_power_meter_modbus_read.system_frequency;



opc.popa_supervisor_kt_2720_line_to_neutral_voltage_scaled_value := modbus_mapping.ro_power_meter_modbus_read.avg_line_to_neutral_voltage;

opc.popa_supervisor_kt_2720_line_to_line_voltage_scaled_value := modbus_mapping.ro_power_meter_modbus_read.avg_line_to_line_voltage;

opc.popa_supervisor_kt_2720_avg_line_current_scaled_value := modbus_mapping.ro_power_meter_modbus_read.system_avg_line_current;

opc.popa_supervisor_kt_2720_total_active_power_scaled_value := modbus_mapping.ro_power_meter_modbus_read.total_active_power;

opc.popa_supervisor_kt_2720_total_reactive_power_scaled_value := modbus_mapping.ro_power_meter_modbus_read.total_reactive_power;

opc.popa_supervisor_kt_2720_total_apparent_power_scaled_value := modbus_mapping.ro_power_meter_modbus_read.total_apparent_power;

opc.popa_supervisor_kt_2720_total_power_factor_scaled_value := modbus_mapping.ro_power_meter_modbus_read.total_power_factor;

opc.popa_supervisor_kt_2720_system_frequency_scaled_value := modbus_mapping.ro_power_meter_modbus_read.system_frequency;


opc.popa_supervisor_kt_2725_line_to_neutral_voltage_scaled_value := modbus_mapping.rocip_power_meter_modbus_read.avg_line_to_neutral_voltage;

opc.popa_supervisor_kt_2725_line_to_line_voltage_scaled_value := modbus_mapping.rocip_power_meter_modbus_read.avg_line_to_line_voltage;

opc.popa_supervisor_kt_2725_avg_line_current_scaled_value := modbus_mapping.rocip_power_meter_modbus_read.system_avg_line_current;

opc.popa_supervisor_kt_2725_total_active_power_scaled_value := modbus_mapping.rocip_power_meter_modbus_read.total_active_power;

opc.popa_supervisor_kt_2725_total_reactive_power_scaled_value := modbus_mapping.rocip_power_meter_modbus_read.total_reactive_power;

opc.popa_supervisor_kt_2725_total_apparent_power_scaled_value := modbus_mapping.rocip_power_meter_modbus_read.total_apparent_power;

opc.popa_supervisor_kt_2725_total_power_factor_scaled_value := modbus_mapping.rocip_power_meter_modbus_read.total_power_factor;

opc.popa_supervisor_kt_2725_system_frequency_scaled_value := modbus_mapping.rocip_power_meter_modbus_read.system_frequency;


opc.popa_supervisor_kt_2730_line_to_neutral_voltage_scaled_value := modbus_mapping.prexfer_power_meter_modbus_read.avg_line_to_neutral_voltage;

opc.popa_supervisor_kt_2730_line_to_line_voltage_scaled_value := modbus_mapping.prexfer_power_meter_modbus_read.avg_line_to_line_voltage;

opc.popa_supervisor_kt_2730_avg_line_current_scaled_value := modbus_mapping.prexfer_power_meter_modbus_read.system_avg_line_current;

opc.popa_supervisor_kt_2730_total_active_power_scaled_value := modbus_mapping.prexfer_power_meter_modbus_read.total_active_power;

opc.popa_supervisor_kt_2730_total_reactive_power_scaled_value := modbus_mapping.prexfer_power_meter_modbus_read.total_reactive_power;

opc.popa_supervisor_kt_2730_total_apparent_power_scaled_value := modbus_mapping.prexfer_power_meter_modbus_read.total_apparent_power;

opc.popa_supervisor_kt_2730_total_power_factor_scaled_value := modbus_mapping.prexfer_power_meter_modbus_read.total_power_factor;

opc.popa_supervisor_kt_2730_system_frequency_scaled_value := modbus_mapping.prexfer_power_meter_modbus_read.system_frequency;


opc.popa_supervisor_kt_3720_line_to_neutral_voltage_scaled_value := modbus_mapping.bop_power_meter_modbus_read.avg_line_to_neutral_voltage;

opc.popa_supervisor_kt_3720_line_to_line_voltage_scaled_value := modbus_mapping.bop_power_meter_modbus_read.avg_line_to_line_voltage;

opc.popa_supervisor_kt_3720_avg_line_current_scaled_value := modbus_mapping.bop_power_meter_modbus_read.system_avg_line_current;

opc.popa_supervisor_kt_3720_total_active_power_scaled_value := modbus_mapping.bop_power_meter_modbus_read.total_active_power;

opc.popa_supervisor_kt_3720_total_reactive_power_scaled_value := modbus_mapping.bop_power_meter_modbus_read.total_reactive_power;

opc.popa_supervisor_kt_3720_total_apparent_power_scaled_value := modbus_mapping.bop_power_meter_modbus_read.total_apparent_power;

opc.popa_supervisor_kt_3720_total_power_factor_scaled_value := modbus_mapping.bop_power_meter_modbus_read.total_power_factor;

opc.popa_supervisor_kt_3720_system_frequency_scaled_value := modbus_mapping.bop_power_meter_modbus_read.system_frequency;


opc.popa_supervisor_kt_1720_line_to_neutral_voltage_scaled_value := modbus_mapping.prodxfer_power_meter_modbus_read.avg_line_to_neutral_voltage;

opc.popa_supervisor_kt_1720_line_to_line_voltage_scaled_value := modbus_mapping.prodxfer_power_meter_modbus_read.avg_line_to_line_voltage;

opc.popa_supervisor_kt_1720_avg_line_current_scaled_value := modbus_mapping.prodxfer_power_meter_modbus_read.system_avg_line_current;

opc.popa_supervisor_kt_1720_total_active_power_scaled_value := modbus_mapping.prodxfer_power_meter_modbus_read.total_active_power;

opc.popa_supervisor_kt_1720_total_reactive_power_scaled_value := modbus_mapping.prodxfer_power_meter_modbus_read.total_reactive_power;

opc.popa_supervisor_kt_1720_total_apparent_power_scaled_value := modbus_mapping.prodxfer_power_meter_modbus_read.total_apparent_power;

opc.popa_supervisor_kt_1720_total_power_factor_scaled_value := modbus_mapping.prodxfer_power_meter_modbus_read.total_power_factor;

opc.popa_supervisor_kt_1720_system_frequency_scaled_value := modbus_mapping.prodxfer_power_meter_modbus_read.system_frequency;


opc.popa_supervisor_kt_4710_line_to_neutral_voltage_scaled_value := modbus_mapping.acid_power_meter_modbus_read.avg_line_to_neutral_voltage;

opc.popa_supervisor_kt_4710_line_to_line_voltage_scaled_value := modbus_mapping.acid_power_meter_modbus_read.avg_line_to_line_voltage;

opc.popa_supervisor_kt_4710_avg_line_current_scaled_value := modbus_mapping.acid_power_meter_modbus_read.system_avg_line_current;

opc.popa_supervisor_kt_4710_total_active_power_scaled_value := modbus_mapping.acid_power_meter_modbus_read.total_active_power;

opc.popa_supervisor_kt_4710_total_reactive_power_scaled_value := modbus_mapping.acid_power_meter_modbus_read.total_reactive_power;

opc.popa_supervisor_kt_4710_total_apparent_power_scaled_value := modbus_mapping.acid_power_meter_modbus_read.total_apparent_power;

opc.popa_supervisor_kt_4710_total_power_factor_scaled_value := modbus_mapping.acid_power_meter_modbus_read.total_power_factor;

opc.popa_supervisor_kt_4710_system_frequency_scaled_value := modbus_mapping.acid_power_meter_modbus_read.system_frequency;


opc.popa_supervisor_kt_1725_line_to_neutral_voltage_scaled_value := modbus_mapping.barge_power_meter_modbus_read.avg_line_to_neutral_voltage;

opc.popa_supervisor_kt_1725_line_to_line_voltage_scaled_value := modbus_mapping.barge_power_meter_modbus_read.avg_line_to_line_voltage;

opc.popa_supervisor_kt_1725_avg_line_current_scaled_value := modbus_mapping.barge_power_meter_modbus_read.system_avg_line_current;

opc.popa_supervisor_kt_1725_total_active_power_scaled_value := modbus_mapping.barge_power_meter_modbus_read.total_active_power;

opc.popa_supervisor_kt_1725_total_reactive_power_scaled_value := modbus_mapping.barge_power_meter_modbus_read.total_reactive_power;

opc.popa_supervisor_kt_1725_total_apparent_power_scaled_value := modbus_mapping.barge_power_meter_modbus_read.total_apparent_power;

opc.popa_supervisor_kt_1725_total_power_factor_scaled_value := modbus_mapping.barge_power_meter_modbus_read.total_power_factor;

opc.popa_supervisor_kt_1725_system_frequency_scaled_value := modbus_mapping.barge_power_meter_modbus_read.system_frequency;


opc.popa_supervisor_kt_1715_line_to_neutral_voltage_scaled_value := modbus_mapping.electrical_shed_power_meter.avg_line_to_neutral_voltage;

opc.popa_supervisor_kt_1715_line_to_line_voltage_scaled_value := modbus_mapping.electrical_shed_power_meter.avg_line_to_line_voltage;

opc.popa_supervisor_kt_1715_avg_line_current_scaled_value := modbus_mapping.electrical_shed_power_meter.system_avg_line_current;

opc.popa_supervisor_kt_1715_total_active_power_scaled_value := modbus_mapping.electrical_shed_power_meter.total_active_power;

opc.popa_supervisor_kt_1715_total_reactive_power_scaled_value := modbus_mapping.electrical_shed_power_meter.total_reactive_power;

opc.popa_supervisor_kt_1715_total_apparent_power_scaled_value := modbus_mapping.electrical_shed_power_meter.total_apparent_power;

opc.popa_supervisor_kt_1715_total_power_factor_scaled_value := modbus_mapping.electrical_shed_power_meter.total_power_factor;

opc.popa_supervisor_kt_1715_system_frequency_scaled_value := modbus_mapping.electrical_shed_power_meter.system_frequency;

opc.popa_supervisor_kt_1715_ground_current_scaled_value := modbus_mapping.electrical_shed_power_meter.ground_current;

opc.popa_supervisor_kt_1715_current_capacity_scaled_value := modbus_mapping.electrical_shed_power_meter.avg_current_capacity;

opc.popa_supervisor_kt_1715_power_factor_leading_scaled_value := modbus_mapping.electrical_shed_power_meter.power_factor_leading;

opc.popa_supervisor_kt_1715_power_factor_lagging_scaled_value := modbus_mapping.electrical_shed_power_meter.power_factor_lagging;



opc.popa_supervisor_kt_1710_line_to_neutral_voltage_scaled_value := modbus_mapping.electrical_bunker_power_meter.avg_line_to_neutral_voltage;

opc.popa_supervisor_kt_1710_line_to_line_voltage_scaled_value := modbus_mapping.electrical_bunker_power_meter.avg_line_to_line_voltage;

opc.popa_supervisor_kt_1710_avg_line_current_scaled_value := modbus_mapping.electrical_bunker_power_meter.system_avg_line_current;

opc.popa_supervisor_kt_1710_total_active_power_scaled_value := modbus_mapping.electrical_bunker_power_meter.total_active_power;

opc.popa_supervisor_kt_1710_total_reactive_power_scaled_value := modbus_mapping.electrical_bunker_power_meter.total_reactive_power;

opc.popa_supervisor_kt_1710_total_apparent_power_scaled_value := modbus_mapping.electrical_bunker_power_meter.total_apparent_power;

opc.popa_supervisor_kt_1710_total_power_factor_scaled_value := modbus_mapping.electrical_bunker_power_meter.total_power_factor;

opc.popa_supervisor_kt_1710_system_frequency_scaled_value := modbus_mapping.electrical_bunker_power_meter.system_frequency;

opc.popa_supervisor_kt_1710_ground_current_scaled_value := modbus_mapping.electrical_bunker_power_meter.ground_current;

opc.popa_supervisor_kt_1710_current_capacity_scaled_value := modbus_mapping.electrical_bunker_power_meter.avg_current_capacity;

opc.popa_supervisor_kt_1710_power_factor_leading_scaled_value := modbus_mapping.electrical_bunker_power_meter.power_factor_leading;

opc.popa_supervisor_kt_1710_power_factor_lagging_scaled_value := modbus_mapping.electrical_bunker_power_meter.power_factor_lagging;

END_PROGRAM

// ---- POUs/heartbeat_routine.TcPOU
PROGRAM heartbeat_routine
VAR
	opc_heartbeat_error : BOOL;
	heartbeat_ton: TON;
	heartbeat_delay_ton: TON;
	heartbeat_alm_ton: TON;
END_VAR

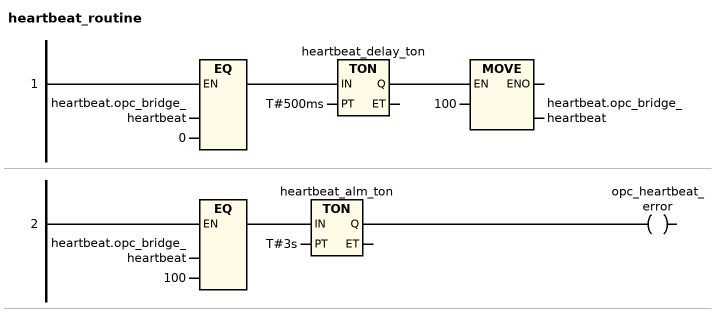
// NETWORK 1
heartbeat_delay_ton(IN := heartbeat.opc_bridge_heartbeat = 0, PT := T#500ms); // TON
IF heartbeat_delay_ton.Q THEN heartbeat.opc_bridge_heartbeat := 100; END_IF

// NETWORK 2
heartbeat_alm_ton(IN := heartbeat.opc_bridge_heartbeat = 100, PT := T#3s); // TON
opc_heartbeat_error := heartbeat_alm_ton.Q;

END_PROGRAM

// ---- POUs/eap_mapping.TcPOU
PROGRAM eap_mapping
VAR
//--- EAP Mapping should be done at the device level - mapping should not need to change after creation -----------
	//--- Inputs --------------------------------------------------------------------------------------------------	
	
	barge_warning_alarm AT %I* : BOOL;
	barge_error_alarm AT %I* : BOOL;
	barge_critical_alarm AT %I* : BOOL;
	
	prodxfer_warning_alarm AT %I* : BOOL;
	prodxfer_error_alarm AT %I* : BOOL;
	prodxfer_critical_alarm AT %I* : BOOL;
	
	acid_warning_alarm AT %I* : BOOL;
	acid_error_alarm AT %I* : BOOL;
	acid_critical_alarm AT %I* : BOOL;
	
	ed_warning_alarm AT %I* : BOOL;
	ed_error_alarm AT %I* : BOOL;
	ed_critical_alarm AT %I* : BOOL;
	
	prexfer_warning_alarm AT %I* : BOOL;
	prexfer_error_alarm AT %I* : BOOL;
	prexfer_critical_alarm AT %I* : BOOL;
	
	//--- Outputs -------------------------------------------------------------------------------------------------

	sup_barge_warning_alarm AT %Q* : BOOL;
	sup_barge_error_alarm AT %Q* : BOOL;
	sup_barge_critical_alarm AT %Q* : BOOL;
	
	sup_prodxfer_warning_alarm AT %Q* : BOOL;
	sup_prodxfer_error_alarm AT %Q* : BOOL;
	sup_prodxfer_critical_alarm AT %Q* : BOOL;
	
	sup_acid_warning_alarm AT %Q* : BOOL;
	sup_acid_error_alarm AT %Q* : BOOL;
	sup_acid_critical_alarm AT %Q* : BOOL;
	
	sup_ed_warning_alarm AT %Q* : BOOL;
	sup_ed_error_alarm AT %Q* : BOOL;
	sup_ed_critical_alarm AT %Q* : BOOL;
	
	sup_prexfer_warning_alarm AT %Q* : BOOL;
	sup_prexfer_error_alarm AT %Q* : BOOL;
	sup_prexfer_critical_alarm AT %Q* : BOOL;
	
	
	
END_VAR

sup_barge_warning_alarm := alarm_manager.warning_alarm_active;
sup_barge_error_alarm := alarm_manager.error_alarm_active;
sup_barge_critical_alarm := alarm_manager.critical_alarm_active;
	
sup_prodxfer_warning_alarm := alarm_manager.warning_alarm_active;
sup_prodxfer_error_alarm := alarm_manager.error_alarm_active;
sup_prodxfer_critical_alarm := alarm_manager.critical_alarm_active;
	
sup_acid_warning_alarm := alarm_manager.warning_alarm_active;
sup_acid_error_alarm := alarm_manager.error_alarm_active;
sup_acid_critical_alarm := alarm_manager.critical_alarm_active;
	
sup_ed_warning_alarm := alarm_manager.warning_alarm_active;
sup_ed_error_alarm := alarm_manager.error_alarm_active;
sup_ed_critical_alarm := alarm_manager.critical_alarm_active;
	
sup_prexfer_warning_alarm := alarm_manager.warning_alarm_active;
sup_prexfer_error_alarm := alarm_manager.error_alarm_active;
sup_prexfer_critical_alarm := alarm_manager.critical_alarm_active;

END_PROGRAM

// ---- POUs/alarm_manager.TcPOU
PROGRAM alarm_manager
VAR
	warning_alarm_active : BOOL;
	error_alarm_active : BOOL;
	critical_alarm_active : BOOL;
END_VAR

IF(eap_mapping.barge_warning_alarm AND eap_mapping.prexfer_warning_alarm AND eap_mapping.ed_warning_alarm AND eap_mapping.prodxfer_warning_alarm AND eap_mapping.acid_warning_alarm)
	THEN
	warning_alarm_active := 1;
	ELSE
		warning_alarm_active := 0;
END_IF

IF(eap_mapping.barge_error_alarm AND eap_mapping.prexfer_error_alarm AND eap_mapping.ed_error_alarm AND eap_mapping.prodxfer_error_alarm AND eap_mapping.acid_error_alarm)
	THEN
	error_alarm_active := 1;
	ELSE
		error_alarm_active := 0;
END_IF

//IF(eap_mapping.barge_critical_alarm AND eap_mapping.prexfer_critical_alarm AND eap_mapping.ed_critical_alarm AND eap_mapping.prodxfer_critical_alarm AND eap_mapping.acid_critical_alarm) OR (opc.popa_supervisor_safety_reset)
IF(eap_mapping.barge_critical_alarm AND eap_mapping.prexfer_critical_alarm AND eap_mapping.prodxfer_critical_alarm AND eap_mapping.acid_critical_alarm) OR (opc.popa_supervisor_safety_reset)
	THEN
	
	critical_alarm_active := 1;
	ELSE
		//critical_alarm_active := 0;
		critical_alarm_active := 1;
END_IF

END_PROGRAM

// ---- POUs/modbus_mapping.TcPOU
PROGRAM modbus_mapping
VAR
	bop_power_meter_modbus_read : modbus_analog_read;
	prexfer_power_meter_modbus_read : modbus_analog_read;
	prodxfer_power_meter_modbus_read : modbus_analog_read;
	barge_power_meter_modbus_read : modbus_analog_read;
	acid_power_meter_modbus_read : modbus_analog_read;
	bped_main_power_meter_modbus_read : modbus_analog_read;
	bped_stack_power_meter_modbus_read : modbus_analog_read;
	nf1_power_meter_modbus_read : modbus_analog_read;
	ro_power_meter_modbus_read : modbus_analog_read;
	rocip_power_meter_modbus_read : modbus_analog_read;
	nf2_power_meter_modbus_read : modbus_analog_read;
	electrical_shed_power_meter: schneider_modbus_read;
	electrical_bunker_power_meter: schneider_modbus_read;
END_VAR

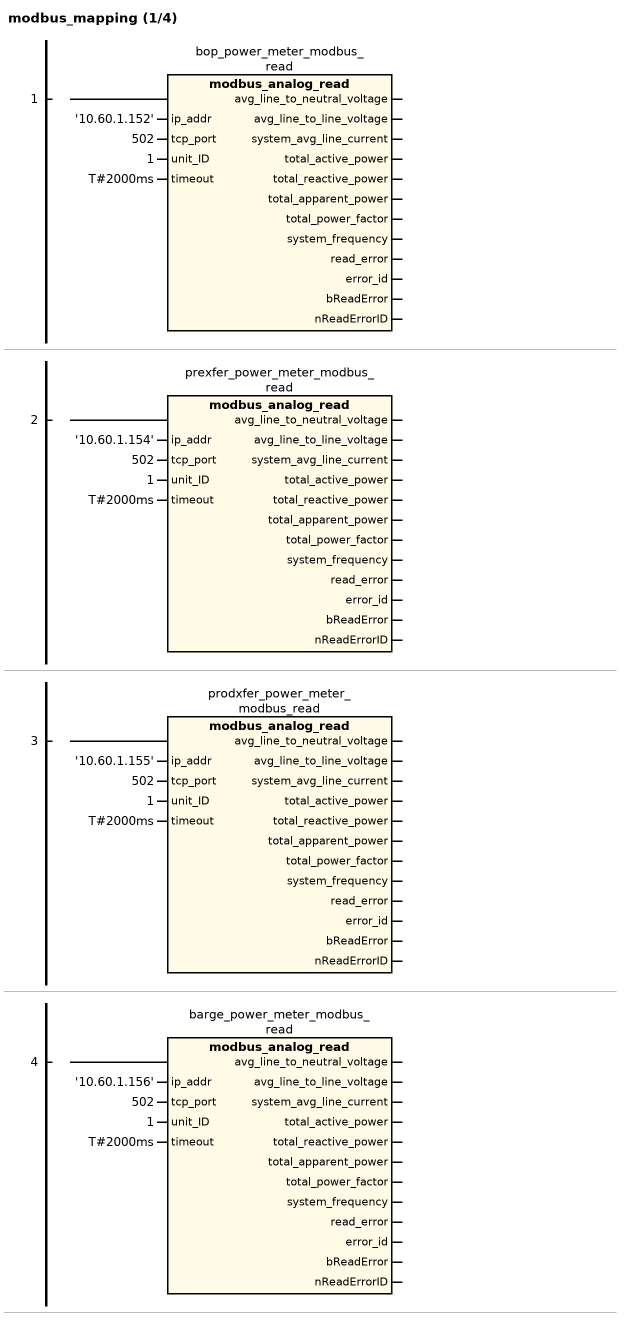
// NETWORK 1
bop_power_meter_modbus_read(ip_addr := '10.60.1.152', tcp_port := 502, unit_ID := 1, timeout := T#2000ms); // modbus_analog_read

// NETWORK 2
prexfer_power_meter_modbus_read(ip_addr := '10.60.1.154', tcp_port := 502, unit_ID := 1, timeout := T#2000ms); // modbus_analog_read

// NETWORK 3
prodxfer_power_meter_modbus_read(
    ip_addr := '10.60.1.155',
    tcp_port := 502,
    unit_ID := 1,
    timeout := T#2000ms); // modbus_analog_read

// NETWORK 4
barge_power_meter_modbus_read(ip_addr := '10.60.1.156', tcp_port := 502, unit_ID := 1, timeout := T#2000ms); // modbus_analog_read

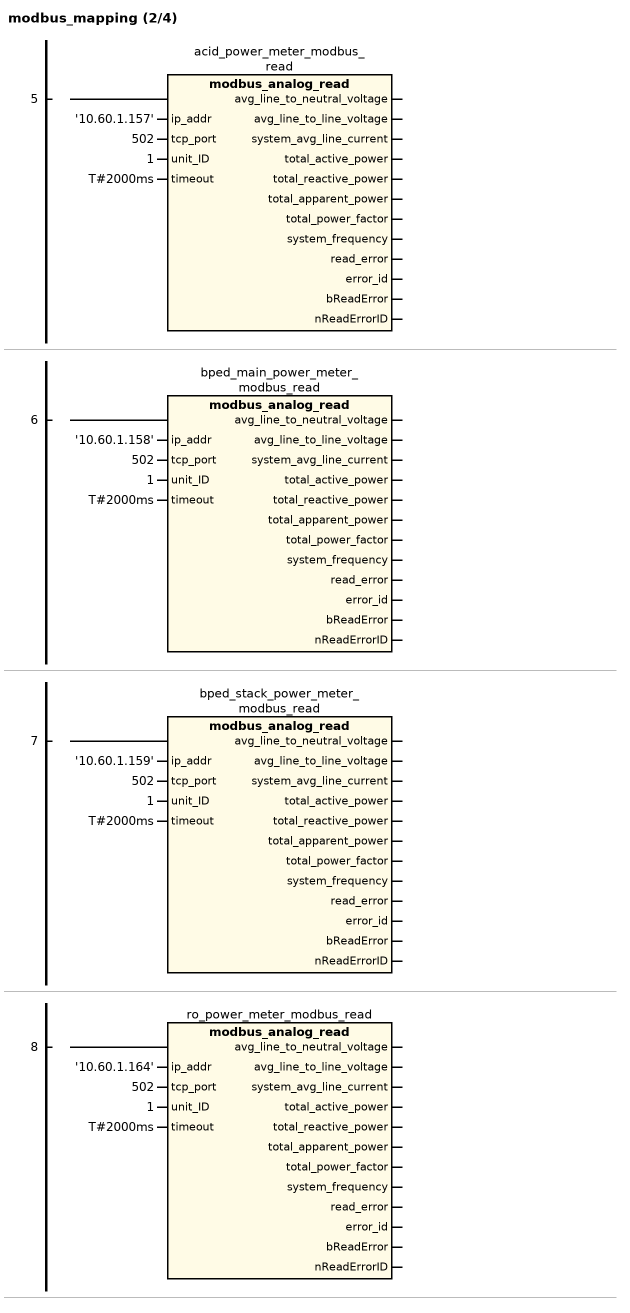
// NETWORK 5
acid_power_meter_modbus_read(ip_addr := '10.60.1.157', tcp_port := 502, unit_ID := 1, timeout := T#2000ms); // modbus_analog_read

// NETWORK 6
bped_main_power_meter_modbus_read(
    ip_addr := '10.60.1.158',
    tcp_port := 502,
    unit_ID := 1,
    timeout := T#2000ms); // modbus_analog_read

// NETWORK 7
bped_stack_power_meter_modbus_read(
    ip_addr := '10.60.1.159',
    tcp_port := 502,
    unit_ID := 1,
    timeout := T#2000ms); // modbus_analog_read

// NETWORK 8
ro_power_meter_modbus_read(ip_addr := '10.60.1.164', tcp_port := 502, unit_ID := 1, timeout := T#2000ms); // modbus_analog_read

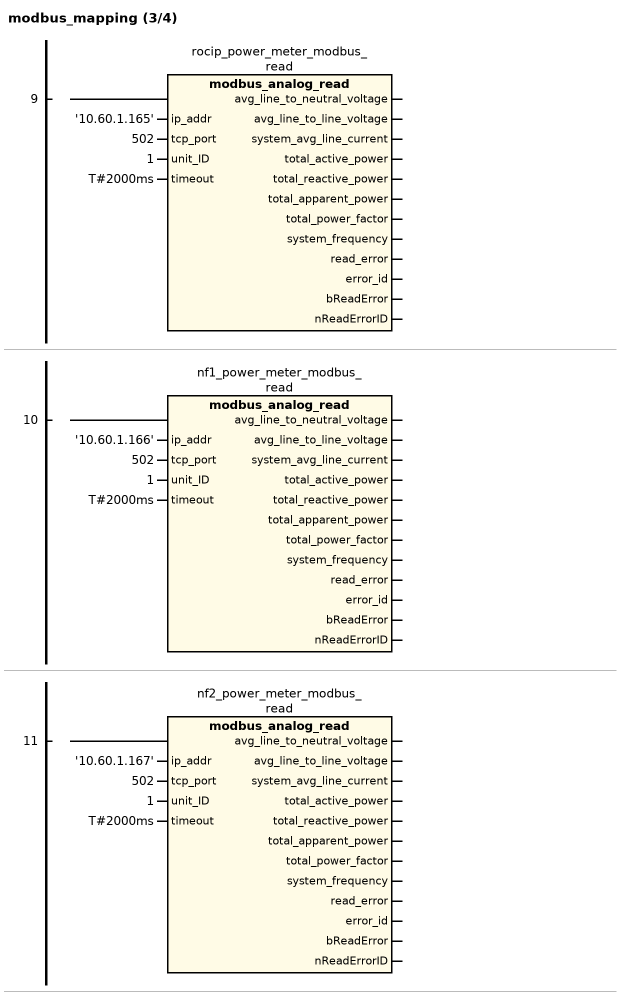
// NETWORK 9
rocip_power_meter_modbus_read(ip_addr := '10.60.1.165', tcp_port := 502, unit_ID := 1, timeout := T#2000ms); // modbus_analog_read

// NETWORK 10
nf1_power_meter_modbus_read(ip_addr := '10.60.1.166', tcp_port := 502, unit_ID := 1, timeout := T#2000ms); // modbus_analog_read

// NETWORK 11
nf2_power_meter_modbus_read(ip_addr := '10.60.1.167', tcp_port := 502, unit_ID := 1, timeout := T#2000ms); // modbus_analog_read

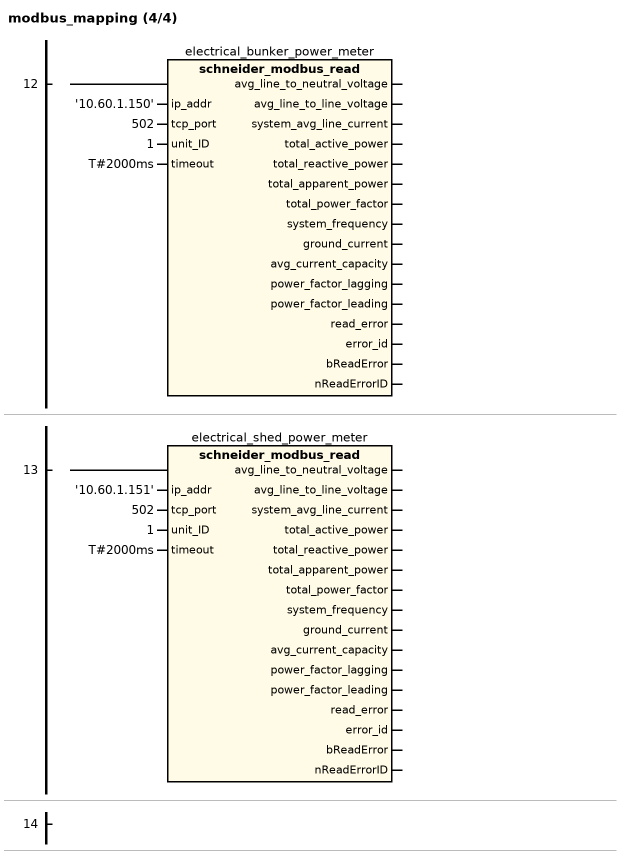
// NETWORK 12
electrical_bunker_power_meter(ip_addr := '10.60.1.150', tcp_port := 502, unit_ID := 1, timeout := T#2000ms); // schneider_modbus_read

// NETWORK 13
electrical_shed_power_meter(ip_addr := '10.60.1.151', tcp_port := 502, unit_ID := 1, timeout := T#2000ms); // schneider_modbus_read

// NETWORK 14

END_PROGRAM

// ---- POUs/Function Blocks/modbus_analog_read.TcPOU
FUNCTION_BLOCK modbus_analog_read
VAR_INPUT
	
	ip_addr : STRING;
	tcp_port : WORD;
	unit_ID : BYTE;

	
	timeout: TIME := T#2000MS;
END_VAR
VAR_OUTPUT
	avg_line_to_neutral_voltage	 : REAL;
	avg_line_to_line_voltage	 : REAL;
	system_avg_line_current	 : REAL;
	total_active_power	 : REAL;
	total_reactive_power	 : REAL;
	total_apparent_power	 : REAL;
	total_power_factor	 : REAL;
	system_frequency	 : REAL;



	read_error : BOOL;
	error_id : UDINT;
	bReadError : BOOL;
	nReadErrorID : UDINT;
END_VAR
VAR
	modbusReadReg : FB_MBReadRegs;
	read_reg : BOOL := TRUE;
	read_regQty : WORD := 16 ;
	reg_address : WORD;
	arrayReadDataReg : ARRAY[0..16] OF WORD;
	msb_hex : STRING; //Modbus register_1 converted word to hex
	lsb_hex : STRING; //Modbus register_2 converted word to hex
	concat_hex : STRING; // hex string concatenated together
	

	avg_line_to_neutral_convert : int_arr_to_real;
	avg_line_to_line_voltage_convert : int_arr_to_real;
	system_avg_line_current_convert : int_arr_to_real;
	total_active_power_convert : int_arr_to_real;
	total_reactive_power_convert : int_arr_to_real;
	total_apparent_power_convert : int_arr_to_real;
	total_power_factor_convert : int_arr_to_real;
	system_frequency_convert : int_arr_to_real;
	

	
	
	read_frequency : TON;
	read_exec : BOOL;
	read_pause : TON;
	count : INT;
	
	cbData: INT;
END_VAR

read_frequency();
read_pause();
read_pause.PT := T#100MS;
read_frequency.PT := T#200MS;
IF read_reg 
THEN
	IF (read_frequency.Q = 0) AND (read_pause.Q = 0)
		THEN
			read_frequency.IN := TRUE;
			read_exec := TRUE;
	ELSIF read_frequency.Q AND (read_pause.Q = 0)
		THEN
			read_exec := FALSE;
			read_pause.IN := TRUE;
	ELSIF read_frequency.Q AND read_pause.Q
		THEN
			read_frequency.IN := FALSE;
			read_pause.IN := FALSE;
			read_exec := FALSE;	
			count:= count + 1;
	END_IF;
END_IF;

IF count > 1
	THEN
	count := 0;
END_IF

CASE count OF
	1:
		reg_address := 27136;
		modbusReadReg(
			sIPAddr:= ip_addr, 
			nTCPPort:= tcp_port, 
			nUnitID:= unit_ID, 
			nQuantity:= read_regQty, 
			nMBAddr:= reg_address, 
			cbLength:= SIZEOF(arrayReadDataReg), 
			pDestAddr:= ADR(arrayReadDataReg), 
			bExecute:= read_frequency.Q, 
			tTimeout:= timeout, 
			bBusy=> , 
			bError=> read_error, 
			nErrId=> error_id, 
			cbRead=> 
		);

	avg_line_to_neutral_convert(array_pos_0 := arrayReadDataReg[0], array_pos_1 := arrayReadDataReg[1], output => avg_line_to_neutral_voltage);
	avg_line_to_line_voltage_convert(array_pos_0 := arrayReadDataReg[2], array_pos_1 := arrayReadDataReg[3], output => avg_line_to_line_voltage);
	system_avg_line_current_convert(array_pos_0 := arrayReadDataReg[4], array_pos_1 := arrayReadDataReg[5], output => system_avg_line_current);
	total_active_power_convert(array_pos_0 := arrayReadDataReg[6], array_pos_1 := arrayReadDataReg[7], output => total_active_power);
	total_reactive_power_convert(array_pos_0 := arrayReadDataReg[8], array_pos_1 := arrayReadDataReg[9], output => total_reactive_power);
	total_apparent_power_convert(array_pos_0 := arrayReadDataReg[10], array_pos_1 := arrayReadDataReg[11], output => total_apparent_power);
	total_power_factor_convert(array_pos_0 := arrayReadDataReg[12], array_pos_1 := arrayReadDataReg[13], output => total_power_factor);
	system_frequency_convert(array_pos_0 := arrayReadDataReg[14], array_pos_1 := arrayReadDataReg[15], output => system_frequency);
(*	avg_line_to_neutral_convert()	 := arrayReadDataReg[0];
	avg_line_to_line_voltage	 := arrayReadDataReg[1];
	system_avg_line_current	 := arrayReadDataReg[2];
	total_active_power	 := arrayReadDataReg[3];
	total_reactive_power	 := arrayReadDataReg[4];
	total_apparent_power	 := arrayReadDataReg[5];
	total_power_factor	 := arrayReadDataReg[6];
	system_frequency	 := arrayReadDataReg[7];
	*)		
//		END_IF
(*		
		temp_output := temp_uconvert.rReal;
	2:
		reg_address := depth_reg_address;
		modbusReadReg(
			sIPAddr:= ip_addr, 
			nTCPPort:= tcp_port, 
			nUnitID:= unit_ID, 
			nQuantity:= read_regQty, 
			nMBAddr:= reg_address, 
			cbLength:= SIZEOF(depth_arrayReadDataReg), 
			pDestAddr:= ADR(depth_arrayReadDataReg), 
			bExecute:= read_frequency.Q, 
			tTimeout:= timeout, 
			bBusy=> , 
			bError=> read_error, 
			nErrId=> error_id, 
			cbRead=> 
		);
	//	IF NOT (depth_read_error)
//			THEN
			//depth_arrayReadDataReg := arrayReadDataReg;
			depth_msb_hex := WORD_TO_HEXSTR(in:= depth_arrayReadDataReg[0], iPrecision:= 4, bLoCase:= FALSE);
			depth_lsb_hex := WORD_TO_HEXSTR(in:= depth_arrayReadDataReg[1], iPrecision:= 4, bLoCase:= FALSE);	
			depth_concat_hex := CONCAT(STR1:=depth_msb_hex , STR2:=depth_lsb_hex );
			depth_cbData := HEXSTR_TO_DATA( depth_concat_hex, ADR( depth_hex_byte_data), SIZEOF( depth_hex_byte_data ) );
			
			depth_uconvert.arrUDP_Data[3] := depth_hex_byte_data[0];
			depth_uconvert.arrUDP_Data[2] := depth_hex_byte_data[1];
			depth_uconvert.arrUDP_Data[1] := depth_hex_byte_data[2];
			depth_uconvert.arrUDP_Data[0] := depth_hex_byte_data[3];
//		END_IF

		
		depth_output := depth_uconvert.rReal;
	3:
		reg_address := conductivity_reg_address;
		modbusReadReg(
			sIPAddr:= ip_addr, 
			nTCPPort:= tcp_port, 
			nUnitID:= unit_ID, 
			nQuantity:= read_regQty, 
			nMBAddr:= reg_address, 
			cbLength:= SIZEOF(conductivity_arrayReadDataReg), 
			pDestAddr:= ADR(conductivity_arrayReadDataReg), 
			bExecute:= read_frequency.Q, 
			tTimeout:= timeout, 
			bBusy=> , 
			bError=> read_error, 
			nErrId=> error_id, 
			cbRead=> 
		);
//		IF NOT (conductivity_read_error)
//			THEN
			//conductivity_arrayReadDataReg := arrayReadDataReg;
			conductivity_msb_hex := WORD_TO_HEXSTR(in:= conductivity_arrayReadDataReg[0], iPrecision:= 4, bLoCase:= FALSE);
			conductivity_lsb_hex := WORD_TO_HEXSTR(in:= conductivity_arrayReadDataReg[1], iPrecision:= 4, bLoCase:= FALSE);	
			conductivity_concat_hex := CONCAT(STR1:=conductivity_msb_hex , STR2:=conductivity_lsb_hex );
			conductivity_cbData := HEXSTR_TO_DATA( conductivity_concat_hex, ADR( conductivity_hex_byte_data), SIZEOF( conductivity_hex_byte_data ) );
			
			conductivity_uconvert.arrUDP_Data[3] := conductivity_hex_byte_data[0];
			conductivity_uconvert.arrUDP_Data[2] := conductivity_hex_byte_data[1];
			conductivity_uconvert.arrUDP_Data[1] := conductivity_hex_byte_data[2];
			conductivity_uconvert.arrUDP_Data[0] := conductivity_hex_byte_data[3];
//		END_IF
		
		
		conductivity_output := conductivity_uconvert.rReal;
	4:
		reg_address := do_reg_address;
		modbusReadReg(
			sIPAddr:= ip_addr, 
			nTCPPort:= tcp_port, 
			nUnitID:= unit_ID, 
			nQuantity:= read_regQty, 
			nMBAddr:= reg_address, 
			cbLength:= SIZEOF(do_arrayReadDataReg), 
			pDestAddr:= ADR(do_arrayReadDataReg), 
			bExecute:= read_frequency.Q, 
			tTimeout:= timeout, 
			bBusy=> , 
			bError=> read_error, 
			nErrId=> error_id, 
			cbRead=> 
		);
	//	IF NOT (do_read_error)
//			THEN
			//do_arrayReadDataReg := arrayReadDataReg;
			do_msb_hex := WORD_TO_HEXSTR(in:= do_arrayReadDataReg[0], iPrecision:= 4, bLoCase:= FALSE);
			do_lsb_hex := WORD_TO_HEXSTR(in:= do_arrayReadDataReg[1], iPrecision:= 4, bLoCase:= FALSE);	
			do_concat_hex := CONCAT(STR1:=do_msb_hex , STR2:=do_lsb_hex );
			do_cbData := HEXSTR_TO_DATA( do_concat_hex, ADR( do_hex_byte_data), SIZEOF( do_hex_byte_data ) );
			
			do_uconvert.arrUDP_Data[3] := do_hex_byte_data[0];
			do_uconvert.arrUDP_Data[2] := do_hex_byte_data[1];
			do_uconvert.arrUDP_Data[1] := do_hex_byte_data[2];
			do_uconvert.arrUDP_Data[0] := do_hex_byte_data[3];
//		END_IF
		
		
		do_output := do_uconvert.rReal;
	5:
		reg_address := ph_reg_address;
		modbusReadReg(
			sIPAddr:= ip_addr, 
			nTCPPort:= tcp_port, 
			nUnitID:= unit_ID, 
			nQuantity:= read_regQty, 
			nMBAddr:= reg_address, 
			cbLength:= SIZEOF(ph_arrayReadDataReg), 
			pDestAddr:= ADR(ph_arrayReadDataReg), 
			bExecute:= read_frequency.Q, 
			tTimeout:= timeout, 
			bBusy=> , 
			bError=> read_error, 
			nErrId=> error_id, 
			cbRead=> 
		);
	//	IF NOT ph_read_error
	//		THEN
			//ph_arrayReadDataReg := arrayReadDataReg;
			ph_msb_hex := WORD_TO_HEXSTR(in:= ph_arrayReadDataReg[0], iPrecision:= 4, bLoCase:= FALSE);
			ph_lsb_hex := WORD_TO_HEXSTR(in:= ph_arrayReadDataReg[1], iPrecision:= 4, bLoCase:= FALSE);	
			ph_concat_hex := CONCAT(STR1:=ph_msb_hex , STR2:=ph_lsb_hex );
			ph_cbData := HEXSTR_TO_DATA( ph_concat_hex, ADR( ph_hex_byte_data), SIZEOF( ph_hex_byte_data ) );
			
			ph_uconvert.arrUDP_Data[3] := ph_hex_byte_data[0];
			ph_uconvert.arrUDP_Data[2] := ph_hex_byte_data[1];
			ph_uconvert.arrUDP_Data[1] := ph_hex_byte_data[2];
			ph_uconvert.arrUDP_Data[0] := ph_hex_byte_data[3];
	//	END_IF
		
		
		ph_output := ph_uconvert.rReal;
	6:
		reg_address := turbidity_reg_address;
		modbusReadReg(
			sIPAddr:= ip_addr, 
			nTCPPort:= tcp_port, 
			nUnitID:= unit_ID, 
			nQuantity:= read_regQty, 
			nMBAddr:= reg_address, 
			cbLength:= SIZEOF(turbidity_arrayReadDataReg), 
			pDestAddr:= ADR(turbidity_arrayReadDataReg), 
			bExecute:= read_frequency.Q, 
			tTimeout:= timeout, 
			bBusy=> , 
			bError=> read_error, 
			nErrId=> error_id, 
			cbRead=> 
		);
	//	IF NOT (turbidity_read_error)
	//		THEN
			//turbidity_arrayReadDataReg := arrayReadDataReg;
			turbidity_msb_hex := WORD_TO_HEXSTR(in:= turbidity_arrayReadDataReg[0], iPrecision:= 4, bLoCase:= FALSE);
			turbidity_lsb_hex := WORD_TO_HEXSTR(in:= turbidity_arrayReadDataReg[1], iPrecision:= 4, bLoCase:= FALSE);	
			turbidity_concat_hex := CONCAT(STR1:=turbidity_msb_hex , STR2:=turbidity_lsb_hex );
			turbidity_cbData := HEXSTR_TO_DATA( turbidity_concat_hex, ADR( turbidity_hex_byte_data), SIZEOF( turbidity_hex_byte_data ) );
			
			turbidity_uconvert.arrUDP_Data[3] := turbidity_hex_byte_data[0];
			turbidity_uconvert.arrUDP_Data[2] := turbidity_hex_byte_data[1];
			turbidity_uconvert.arrUDP_Data[1] := turbidity_hex_byte_data[2];
			turbidity_uconvert.arrUDP_Data[0] := turbidity_hex_byte_data[3];
		
	//	END_IF

		turbidity_output := turbidity_uconvert.rReal;
	7:
		reg_address := voltage_reg_address;
		modbusReadReg(
			sIPAddr:= ip_addr, 
			nTCPPort:= tcp_port, 
			nUnitID:= unit_ID, 
			nQuantity:= read_regQty, 
			nMBAddr:= reg_address, 
			cbLength:= SIZEOF(voltage_arrayReadDataReg), 
			pDestAddr:= ADR(voltage_arrayReadDataReg), 
			bExecute:= read_frequency.Q, 
			tTimeout:= timeout, 
			bBusy=> , 
			bError=> read_error, 
			nErrId=> error_id, 
			cbRead=> 
		);
//		IF NOT (voltage_read_error)
//			THEN
			//voltage_arrayReadDataReg := arrayReadDataReg;
			voltage_msb_hex := WORD_TO_HEXSTR(in:= voltage_arrayReadDataReg[0], iPrecision:= 4, bLoCase:= FALSE);
			voltage_lsb_hex := WORD_TO_HEXSTR(in:= voltage_arrayReadDataReg[1], iPrecision:= 4, bLoCase:= FALSE);	
			voltage_concat_hex := CONCAT(STR1:=voltage_msb_hex , STR2:=voltage_lsb_hex );
			voltage_cbData := HEXSTR_TO_DATA( voltage_concat_hex, ADR( voltage_hex_byte_data), SIZEOF( voltage_hex_byte_data ) );
			
			voltage_uconvert.arrUDP_Data[3] := voltage_hex_byte_data[0];
			voltage_uconvert.arrUDP_Data[2] := voltage_hex_byte_data[1];
			voltage_uconvert.arrUDP_Data[1] := voltage_hex_byte_data[2];
			voltage_uconvert.arrUDP_Data[0] := voltage_hex_byte_data[3];
//		END_IF
		
		
		voltage_output := voltage_uconvert.rReal;
	8:
		reg_address := battery_reg_address;
		modbusReadReg(
			sIPAddr:= ip_addr, 
			nTCPPort:= tcp_port, 
			nUnitID:= unit_ID, 
			nQuantity:= read_regQty, 
			nMBAddr:= reg_address, 
			cbLength:= SIZEOF(battery_arrayReadDataReg), 
			pDestAddr:= ADR(battery_arrayReadDataReg), 
			bExecute:= read_frequency.Q, 
			tTimeout:= timeout, 
			bBusy=> , 
			bError=> read_error, 
			nErrId=> error_id, 
			cbRead=> 
		);
//		IF not battery_read_error
//			THEN
			//battery_arrayReadDataReg := arrayReadDataReg;
			battery_msb_hex := WORD_TO_HEXSTR(in:= battery_arrayReadDataReg[0], iPrecision:= 4, bLoCase:= FALSE);
			battery_lsb_hex := WORD_TO_HEXSTR(in:= battery_arrayReadDataReg[1], iPrecision:= 4, bLoCase:= FALSE);	
			battery_concat_hex := CONCAT(STR1:=battery_msb_hex , STR2:=battery_lsb_hex );
			battery_cbData := HEXSTR_TO_DATA( battery_concat_hex, ADR( battery_hex_byte_data), SIZEOF( battery_hex_byte_data ) );
			
			battery_uconvert.arrUDP_Data[3] := battery_hex_byte_data[0];
			battery_uconvert.arrUDP_Data[2] := battery_hex_byte_data[1];
			battery_uconvert.arrUDP_Data[1] := battery_hex_byte_data[2];
			battery_uconvert.arrUDP_Data[0] := battery_hex_byte_data[3];
	//	END_IF
		
		
		battery_output := battery_uconvert.rReal;
*)	
END_CASE

END_FUNCTION_BLOCK

// ---- POUs/Function Blocks/int_arr_to_real.TcPOU
FUNCTION_BLOCK int_arr_to_real
VAR_INPUT
	array_pos_0 : WORD;
	array_pos_1 : WORD;
END_VAR
VAR_OUTPUT
	output : REAL;
END_VAR
VAR
	msb_hex: STRING(255);
	lsb_hex: STRING(255);
	concat_hex: STRING(255);
	cbData: UDINT;
	hex_byte_data:  ARRAY[0..3] OF BYTE;;
	uConvert : U_Convert;
END_VAR

msb_hex := WORD_TO_HEXSTR(in := array_pos_0, iPrecision := 4, bLoCase := FALSE);
lsb_hex := WORD_TO_HEXSTR(in := array_pos_1, iPrecision := 4, bLoCase := FALSE);	

concat_hex := CONCAT(STR1 := msb_hex , STR2 := lsb_hex );

cbData := HEXSTR_TO_DATA( concat_hex, ADR( hex_byte_data), SIZEOF( hex_byte_data ) );
			
uconvert.arrUDP_Data[3] := hex_byte_data[0];
uconvert.arrUDP_Data[2] := hex_byte_data[1];
uconvert.arrUDP_Data[1] := hex_byte_data[2];
uconvert.arrUDP_Data[0] := hex_byte_data[3];

output := uconvert.rReal;

END_FUNCTION_BLOCK

// ---- POUs/Function Blocks/schneider_modbus_read.TcPOU
FUNCTION_BLOCK schneider_modbus_read
VAR_INPUT
	
	ip_addr : STRING;
	tcp_port : WORD;
	unit_ID : BYTE;

	
	timeout: TIME := T#2000MS;
END_VAR
VAR_OUTPUT
	avg_line_to_neutral_voltage	 : REAL;
	avg_line_to_line_voltage	 : REAL;
	system_avg_line_current	 : REAL;
	total_active_power	 : REAL;
	total_reactive_power	 : REAL;
	total_apparent_power	 : REAL;
	total_power_factor	 : REAL;
	system_frequency	 : REAL;
	ground_current : REAL;
	avg_current_capacity : REAL;
	power_factor_lagging : REAL;
	power_factor_leading : REAL;



	read_error : BOOL;
	error_id : UDINT;
	bReadError : BOOL;
	nReadErrorID : UDINT;
END_VAR
VAR
	modbusReadReg : FB_MBReadRegs;
	read_reg : BOOL := TRUE;
	read_regQty : WORD := 100 ;
	reg_address : WORD;
	arrayReadDataReg_1 : ARRAY[0..100] OF WORD;
	arrayReadDataReg_2 : ARRAY[0..100] OF WORD;
	msb_hex : STRING; //Modbus register_1 converted word to hex
	lsb_hex : STRING; //Modbus register_2 converted word to hex
	concat_hex : STRING; // hex string concatenated together
	

	avg_line_to_neutral_convert : int_arr_to_real;
	avg_line_to_line_voltage_convert : int_arr_to_real;
	system_avg_line_current_convert : int_arr_to_real;
	total_active_power_convert : int_arr_to_real;
	total_reactive_power_convert : int_arr_to_real;
	total_apparent_power_convert : int_arr_to_real;
	total_power_factor_convert : int_arr_to_real;
	system_frequency_convert : int_arr_to_real;
	ground_current_convert : int_arr_to_real;
	avg_current_capacity_convert : int_arr_to_real;
	power_factor_lagging_convert : int_arr_to_real;
	power_factor_leading_convert : int_arr_to_real;

	
	
	read_frequency : TON;
	read_exec : BOOL;
	read_pause : TON;
	count : INT;
	
	cbData: INT;
END_VAR

read_frequency();
read_pause();
read_pause.PT := T#1000MS;
read_frequency.PT := T#200MS;
IF read_reg 
THEN
	IF (read_frequency.Q = 0) AND (read_pause.Q = 0)
		THEN
			read_frequency.IN := TRUE;
			read_exec := TRUE;
	ELSIF read_frequency.Q AND (read_pause.Q = 0)
		THEN
			read_exec := FALSE;
			read_pause.IN := TRUE;
	ELSIF read_frequency.Q AND read_pause.Q
		THEN
			read_frequency.IN := FALSE;
			read_pause.IN := FALSE;
			read_exec := FALSE;	
			count:= count + 1;
	END_IF;
END_IF;

IF count > 2
	THEN
	count := 0;
END_IF

CASE count OF
	1:
		reg_address := 2999; //Subtracting 1 to account for minus offset
		modbusReadReg(
			sIPAddr:= ip_addr, 
			nTCPPort:= tcp_port, 
			nUnitID:= unit_ID, 
			nQuantity:= read_regQty, 
			nMBAddr:= reg_address, 
			cbLength:= SIZEOF(arrayReadDataReg_1), 
			pDestAddr:= ADR(arrayReadDataReg_1), 
			bExecute:= read_frequency.Q, 
			tTimeout:= timeout, 
			bBusy=> , 
			bError=> read_error, 
			nErrId=> error_id, 
			cbRead=> 
		);
	
		ground_current_convert(array_pos_0 := arrayReadDataReg_1[8], array_pos_1 := arrayReadDataReg_1[9], output => ground_current);
		avg_line_to_neutral_convert(array_pos_0 := arrayReadDataReg_1[36], array_pos_1 := arrayReadDataReg_1[37], output => avg_line_to_neutral_voltage);
		avg_line_to_line_voltage_convert(array_pos_0 := arrayReadDataReg_1[26], array_pos_1 := arrayReadDataReg_1[27], output => avg_line_to_line_voltage);
		system_avg_line_current_convert(array_pos_0 := arrayReadDataReg_1[10], array_pos_1 := arrayReadDataReg_1[11], output => system_avg_line_current);
		total_active_power_convert(array_pos_0 := arrayReadDataReg_1[60], array_pos_1 := arrayReadDataReg_1[61], output => total_active_power);
		total_reactive_power_convert(array_pos_0 := arrayReadDataReg_1[68], array_pos_1 := arrayReadDataReg_1[69], output => total_reactive_power);
		total_apparent_power_convert(array_pos_0 := arrayReadDataReg_1[76], array_pos_1 := arrayReadDataReg_1[77], output => total_apparent_power);


		
	
	2:
		reg_address := 3099; //Subtracting 1 to account for minus offset
		modbusReadReg(
			sIPAddr:= ip_addr, 
			nTCPPort:= tcp_port, 
			nUnitID:= unit_ID, 
			nQuantity:= read_regQty, 
			nMBAddr:= reg_address, 
			cbLength:= SIZEOF(arrayReadDataReg_2), 
			pDestAddr:= ADR(arrayReadDataReg_2), 
			bExecute:= read_frequency.Q, 
			tTimeout:= timeout, 
			bBusy=> , 
			bError=> read_error, 
			nErrId=> error_id, 
			cbRead=> 
		);
		total_power_factor_convert(array_pos_0 := arrayReadDataReg_2[50], array_pos_1 := arrayReadDataReg_2[51], output => total_power_factor);
		system_frequency_convert(array_pos_0 := arrayReadDataReg_2[10], array_pos_1 := arrayReadDataReg_2[11], output => system_frequency);
		avg_current_capacity_convert(array_pos_0 := arrayReadDataReg_2[42], array_pos_1 := arrayReadDataReg_2[43], output => avg_current_capacity);
		power_factor_lagging_convert(array_pos_0 := arrayReadDataReg_2[72], array_pos_1 := arrayReadDataReg_2[73], output => power_factor_lagging);
		power_factor_leading_convert(array_pos_0 := arrayReadDataReg_2[74], array_pos_1 := arrayReadDataReg_2[75], output => power_factor_leading);
(*	3:
		reg_address := conductivity_reg_address;
		modbusReadReg(
			sIPAddr:= ip_addr, 
			nTCPPort:= tcp_port, 
			nUnitID:= unit_ID, 
			nQuantity:= read_regQty, 
			nMBAddr:= reg_address, 
			cbLength:= SIZEOF(conductivity_arrayReadDataReg), 
			pDestAddr:= ADR(conductivity_arrayReadDataReg), 
			bExecute:= read_frequency.Q, 
			tTimeout:= timeout, 
			bBusy=> , 
			bError=> read_error, 
			nErrId=> error_id, 
			cbRead=> 
		);
//		IF NOT (conductivity_read_error)
//			THEN
			//conductivity_arrayReadDataReg := arrayReadDataReg;
			conductivity_msb_hex := WORD_TO_HEXSTR(in:= conductivity_arrayReadDataReg[0], iPrecision:= 4, bLoCase:= FALSE);
			conductivity_lsb_hex := WORD_TO_HEXSTR(in:= conductivity_arrayReadDataReg[1], iPrecision:= 4, bLoCase:= FALSE);	
			conductivity_concat_hex := CONCAT(STR1:=conductivity_msb_hex , STR2:=conductivity_lsb_hex );
			conductivity_cbData := HEXSTR_TO_DATA( conductivity_concat_hex, ADR( conductivity_hex_byte_data), SIZEOF( conductivity_hex_byte_data ) );
			
			conductivity_uconvert.arrUDP_Data[3] := conductivity_hex_byte_data[0];
			conductivity_uconvert.arrUDP_Data[2] := conductivity_hex_byte_data[1];
			conductivity_uconvert.arrUDP_Data[1] := conductivity_hex_byte_data[2];
			conductivity_uconvert.arrUDP_Data[0] := conductivity_hex_byte_data[3];
//		END_IF
		
		
		conductivity_output := conductivity_uconvert.rReal;
	4:
		reg_address := do_reg_address;
		modbusReadReg(
			sIPAddr:= ip_addr, 
			nTCPPort:= tcp_port, 
			nUnitID:= unit_ID, 
			nQuantity:= read_regQty, 
			nMBAddr:= reg_address, 
			cbLength:= SIZEOF(do_arrayReadDataReg), 
			pDestAddr:= ADR(do_arrayReadDataReg), 
			bExecute:= read_frequency.Q, 
			tTimeout:= timeout, 
			bBusy=> , 
			bError=> read_error, 
			nErrId=> error_id, 
			cbRead=> 
		);
	//	IF NOT (do_read_error)
//			THEN
			//do_arrayReadDataReg := arrayReadDataReg;
			do_msb_hex := WORD_TO_HEXSTR(in:= do_arrayReadDataReg[0], iPrecision:= 4, bLoCase:= FALSE);
			do_lsb_hex := WORD_TO_HEXSTR(in:= do_arrayReadDataReg[1], iPrecision:= 4, bLoCase:= FALSE);	
			do_concat_hex := CONCAT(STR1:=do_msb_hex , STR2:=do_lsb_hex );
			do_cbData := HEXSTR_TO_DATA( do_concat_hex, ADR( do_hex_byte_data), SIZEOF( do_hex_byte_data ) );
			
			do_uconvert.arrUDP_Data[3] := do_hex_byte_data[0];
			do_uconvert.arrUDP_Data[2] := do_hex_byte_data[1];
			do_uconvert.arrUDP_Data[1] := do_hex_byte_data[2];
			do_uconvert.arrUDP_Data[0] := do_hex_byte_data[3];
//		END_IF
		
		
		do_output := do_uconvert.rReal;
	5:
		reg_address := ph_reg_address;
		modbusReadReg(
			sIPAddr:= ip_addr, 
			nTCPPort:= tcp_port, 
			nUnitID:= unit_ID, 
			nQuantity:= read_regQty, 
			nMBAddr:= reg_address, 
			cbLength:= SIZEOF(ph_arrayReadDataReg), 
			pDestAddr:= ADR(ph_arrayReadDataReg), 
			bExecute:= read_frequency.Q, 
			tTimeout:= timeout, 
			bBusy=> , 
			bError=> read_error, 
			nErrId=> error_id, 
			cbRead=> 
		);
	//	IF NOT ph_read_error
	//		THEN
			//ph_arrayReadDataReg := arrayReadDataReg;
			ph_msb_hex := WORD_TO_HEXSTR(in:= ph_arrayReadDataReg[0], iPrecision:= 4, bLoCase:= FALSE);
			ph_lsb_hex := WORD_TO_HEXSTR(in:= ph_arrayReadDataReg[1], iPrecision:= 4, bLoCase:= FALSE);	
			ph_concat_hex := CONCAT(STR1:=ph_msb_hex , STR2:=ph_lsb_hex );
			ph_cbData := HEXSTR_TO_DATA( ph_concat_hex, ADR( ph_hex_byte_data), SIZEOF( ph_hex_byte_data ) );
			
			ph_uconvert.arrUDP_Data[3] := ph_hex_byte_data[0];
			ph_uconvert.arrUDP_Data[2] := ph_hex_byte_data[1];
			ph_uconvert.arrUDP_Data[1] := ph_hex_byte_data[2];
			ph_uconvert.arrUDP_Data[0] := ph_hex_byte_data[3];
	//	END_IF
		
		
		ph_output := ph_uconvert.rReal;
	6:
		reg_address := turbidity_reg_address;
		modbusReadReg(
			sIPAddr:= ip_addr, 
			nTCPPort:= tcp_port, 
			nUnitID:= unit_ID, 
			nQuantity:= read_regQty, 
			nMBAddr:= reg_address, 
			cbLength:= SIZEOF(turbidity_arrayReadDataReg), 
			pDestAddr:= ADR(turbidity_arrayReadDataReg), 
			bExecute:= read_frequency.Q, 
			tTimeout:= timeout, 
			bBusy=> , 
			bError=> read_error, 
			nErrId=> error_id, 
			cbRead=> 
		);
	//	IF NOT (turbidity_read_error)
	//		THEN
			//turbidity_arrayReadDataReg := arrayReadDataReg;
			turbidity_msb_hex := WORD_TO_HEXSTR(in:= turbidity_arrayReadDataReg[0], iPrecision:= 4, bLoCase:= FALSE);
			turbidity_lsb_hex := WORD_TO_HEXSTR(in:= turbidity_arrayReadDataReg[1], iPrecision:= 4, bLoCase:= FALSE);	
			turbidity_concat_hex := CONCAT(STR1:=turbidity_msb_hex , STR2:=turbidity_lsb_hex );
			turbidity_cbData := HEXSTR_TO_DATA( turbidity_concat_hex, ADR( turbidity_hex_byte_data), SIZEOF( turbidity_hex_byte_data ) );
			
			turbidity_uconvert.arrUDP_Data[3] := turbidity_hex_byte_data[0];
			turbidity_uconvert.arrUDP_Data[2] := turbidity_hex_byte_data[1];
			turbidity_uconvert.arrUDP_Data[1] := turbidity_hex_byte_data[2];
			turbidity_uconvert.arrUDP_Data[0] := turbidity_hex_byte_data[3];
		
	//	END_IF

		turbidity_output := turbidity_uconvert.rReal;
	7:
		reg_address := voltage_reg_address;
		modbusReadReg(
			sIPAddr:= ip_addr, 
			nTCPPort:= tcp_port, 
			nUnitID:= unit_ID, 
			nQuantity:= read_regQty, 
			nMBAddr:= reg_address, 
			cbLength:= SIZEOF(voltage_arrayReadDataReg), 
			pDestAddr:= ADR(voltage_arrayReadDataReg), 
			bExecute:= read_frequency.Q, 
			tTimeout:= timeout, 
			bBusy=> , 
			bError=> read_error, 
			nErrId=> error_id, 
			cbRead=> 
		);
//		IF NOT (voltage_read_error)
//			THEN
			//voltage_arrayReadDataReg := arrayReadDataReg;
			voltage_msb_hex := WORD_TO_HEXSTR(in:= voltage_arrayReadDataReg[0], iPrecision:= 4, bLoCase:= FALSE);
			voltage_lsb_hex := WORD_TO_HEXSTR(in:= voltage_arrayReadDataReg[1], iPrecision:= 4, bLoCase:= FALSE);	
			voltage_concat_hex := CONCAT(STR1:=voltage_msb_hex , STR2:=voltage_lsb_hex );
			voltage_cbData := HEXSTR_TO_DATA( voltage_concat_hex, ADR( voltage_hex_byte_data), SIZEOF( voltage_hex_byte_data ) );
			
			voltage_uconvert.arrUDP_Data[3] := voltage_hex_byte_data[0];
			voltage_uconvert.arrUDP_Data[2] := voltage_hex_byte_data[1];
			voltage_uconvert.arrUDP_Data[1] := voltage_hex_byte_data[2];
			voltage_uconvert.arrUDP_Data[0] := voltage_hex_byte_data[3];
//		END_IF
		
		
		voltage_output := voltage_uconvert.rReal;
	8:
		reg_address := battery_reg_address;
		modbusReadReg(
			sIPAddr:= ip_addr, 
			nTCPPort:= tcp_port, 
			nUnitID:= unit_ID, 
			nQuantity:= read_regQty, 
			nMBAddr:= reg_address, 
			cbLength:= SIZEOF(battery_arrayReadDataReg), 
			pDestAddr:= ADR(battery_arrayReadDataReg), 
			bExecute:= read_frequency.Q, 
			tTimeout:= timeout, 
			bBusy=> , 
			bError=> read_error, 
			nErrId=> error_id, 
			cbRead=> 
		);
//		IF not battery_read_error
//			THEN
			//battery_arrayReadDataReg := arrayReadDataReg;
			battery_msb_hex := WORD_TO_HEXSTR(in:= battery_arrayReadDataReg[0], iPrecision:= 4, bLoCase:= FALSE);
			battery_lsb_hex := WORD_TO_HEXSTR(in:= battery_arrayReadDataReg[1], iPrecision:= 4, bLoCase:= FALSE);	
			battery_concat_hex := CONCAT(STR1:=battery_msb_hex , STR2:=battery_lsb_hex );
			battery_cbData := HEXSTR_TO_DATA( battery_concat_hex, ADR( battery_hex_byte_data), SIZEOF( battery_hex_byte_data ) );
			
			battery_uconvert.arrUDP_Data[3] := battery_hex_byte_data[0];
			battery_uconvert.arrUDP_Data[2] := battery_hex_byte_data[1];
			battery_uconvert.arrUDP_Data[1] := battery_hex_byte_data[2];
			battery_uconvert.arrUDP_Data[0] := battery_hex_byte_data[3];
	//	END_IF
		
		
		battery_output := battery_uconvert.rReal;
*)	
END_CASE

END_FUNCTION_BLOCK

// ---- POUs/state_transition.TcPOU
PROGRAM state_transition
VAR PERSISTENT
	//Hard coded state values for comparison
	state_faulted : INT :=0;
	state_stopped : INT :=10;
	state_idle : INT :=20;
	state_cip : INT :=30;
	state_manual : INT :=40;
	state_maint : INT :=50;
	state_active_input : INT :=61;
	state_active_conc : INT :=62;
	state_active_opt : INT :=63;
	
END_VAR

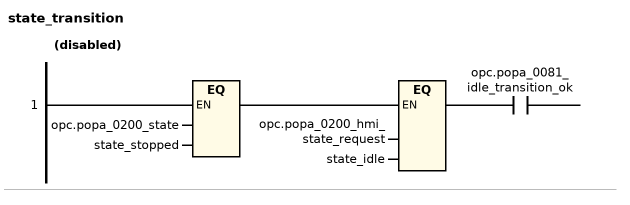
// NETWORK 1 (disabled)
// (* (opc.popa_0200_state = state_stopped AND opc.popa_0200_hmi_state_request = state_idle) AND opc.popa_0081_idle_transition_ok; result not used *)

END_PROGRAM

// ---- POUs/Function Blocks/int_arr_to_real_1.TcPOU
FUNCTION_BLOCK int_arr_to_real_1
VAR_INPUT
	array_pos_0 : WORD;
	array_pos_1 : WORD;
END_VAR
VAR_OUTPUT
	output : REAL;
END_VAR
VAR
	msb_hex: STRING(255);
	lsb_hex: STRING(255);
	concat_hex: STRING(255);
	cbData: UDINT;
	hex_byte_data:  ARRAY[0..3] OF BYTE;;
	uConvert : U_Convert;
END_VAR

msb_hex := WORD_TO_HEXSTR(in := array_pos_0, iPrecision := 4, bLoCase := FALSE);
lsb_hex := WORD_TO_HEXSTR(in := array_pos_1, iPrecision := 4, bLoCase := FALSE);	

concat_hex := CONCAT(STR1 := msb_hex , STR2 := lsb_hex );

cbData := HEXSTR_TO_DATA( concat_hex, ADR( hex_byte_data), SIZEOF( hex_byte_data ) );
			
uconvert.arrUDP_Data[3] := hex_byte_data[0];
uconvert.arrUDP_Data[2] := hex_byte_data[1];
uconvert.arrUDP_Data[1] := hex_byte_data[2];
uconvert.arrUDP_Data[0] := hex_byte_data[3];

output := uconvert.rReal;

END_FUNCTION_BLOCK

// ---- POUs/Function Blocks/motor_starter.TcPOU
FUNCTION_BLOCK Motor_Starter
VAR_INPUT
	//Run Feedback from Motor Starter
	Run_Feedback : BOOL; 
	//Reset trigger for Runtime Maint
	Runtime_Maint_Reset : BOOL;
	//Run Request from PLC Program
	Run_Request : BOOL;
	//Comes from Faults ladder
	Fail_to_Start : BOOL;
	//Comes from faults ladder
	Fail_to_Stop : BOOL;
	//Daily Reset from GENERAL POU
	Daily_Reset : BOOL;
END_VAR
VAR_OUTPUT
	//Tells the motor to start when true, stop when false
	Run_Command : BOOL;
	//Accumulated Runtime Hours Today
	Runtime_Today : REAL;
	//Accumulated Runtime Hours Today
	Runtime_Total : REAL;
	//Resettable Runtime for Maintenance purposes, Description is user adjustable
	Runtime_Maint : REAL;
END_VAR
VAR	
	//Runtime Timer Tags, 1 Minute Timer
	Runtime_TON : TON;
	Runtime_PT : TIME := T#1M;
	Runtime_ET : TIME;
	//Runtime Today Counter
	Runtime_Today_CTU : CTU;
	Runtime_Today_CTU_PV : WORD;
	Runtime_Today_CTU_CV : REAL;
	//Total Runtime Minute Counter
	Runtime_Total_Minute_CTU : CTU;
	Runtime_Total_Minute_CTU_Reset : BOOL;
	Runtime_Total_Minute_CTU_PV : WORD :=60;
	Runtime_Total_Minute_CTU_CV : REAL;
	//Total Runtime Hour Counter
	Runtime_Total_Hour_CTU : CTU;
	Runtime_Total_Hour_CTU_Reset : BOOL;
	Runtime_Total_Hour_CTU_PV : WORD;
	//Maintenance Runtime Minute Counter
	Runtime_Maint_Minute_CTU : CTU;
	Runtime_Maint_Minute_CTU_Reset : BOOL;
	Runtime_Maint_Minute_CTU_PV : WORD :=60;
	Runtime_Maint_Minute_CTU_CV : REAL;
	//Maintenance Runtime Hour Counter
	Runtime_Maint_Hour_CTU : CTU;
	Runtime_Maint_Hour_CTU_PV : WORD;
END_VAR

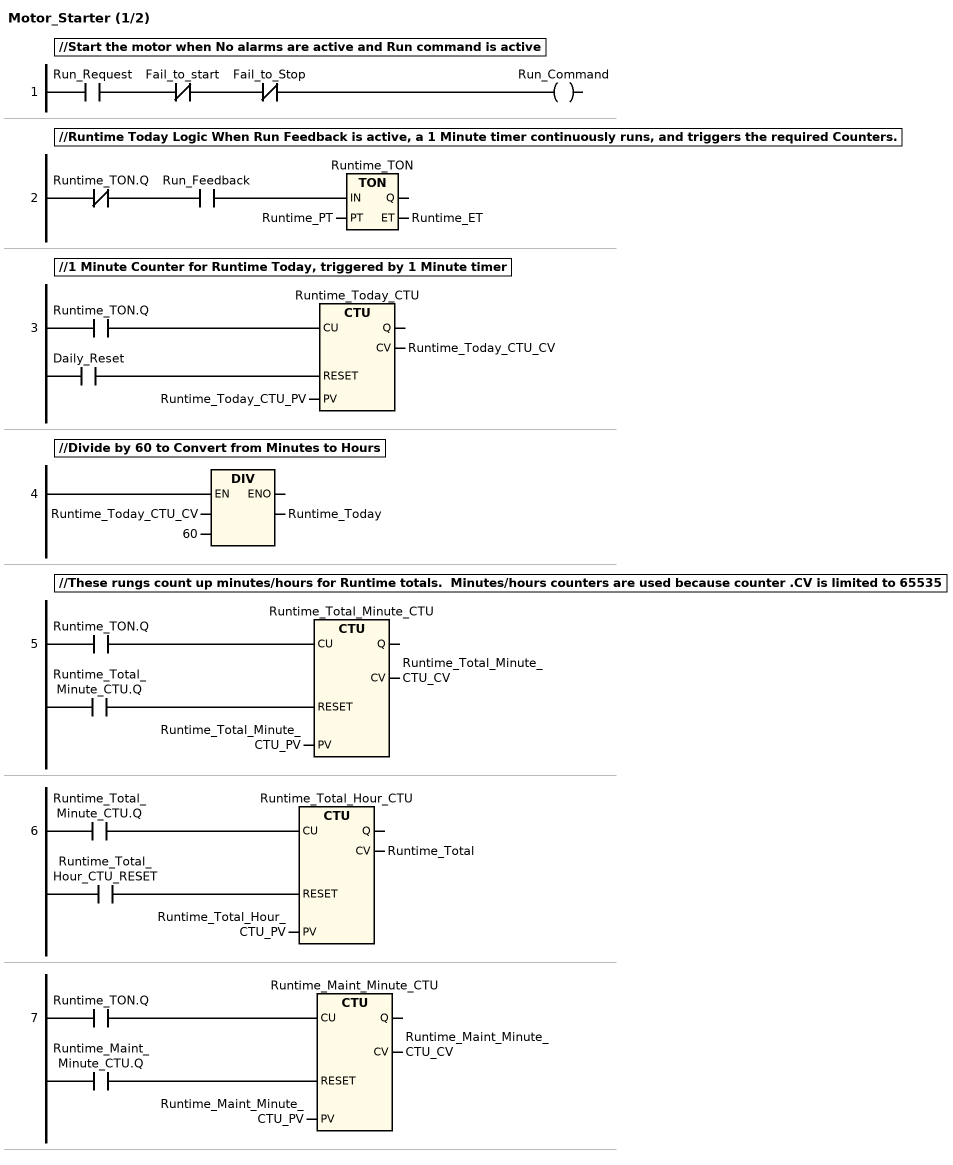
// NETWORK 1
// label: //Start the motor when No alarms are active and Run command is active
Run_Command := Run_Request AND NOT Fail_to_start AND NOT Fail_to_Stop;

// NETWORK 2
// label: //Runtime Today Logic When Run Feedback is active, a 1 Minute timer continuously runs, and triggers the required Counters.
Runtime_TON(IN := NOT Runtime_TON.Q AND Run_Feedback, PT := Runtime_PT, ET => Runtime_ET); // TON

// NETWORK 3
// label: //1 Minute Counter for Runtime Today, triggered by 1 Minute timer
Runtime_Today_CTU(
    CU := Runtime_TON.Q,
    RESET := Daily_Reset,
    PV := Runtime_Today_CTU_PV,
    CV => Runtime_Today_CTU_CV); // CTU

// NETWORK 4
// label: //Divide by 60 to Convert from Minutes to Hours
Runtime_Today := Runtime_Today_CTU_CV / 60;

// NETWORK 5
// label: //These rungs count up minutes/hours for Runtime totals.  Minutes/hours counters are used because counter .CV is limited to 65535
Runtime_Total_Minute_CTU(
    CU := Runtime_TON.Q,
    RESET := Runtime_Total_Minute_CTU.Q,
    PV := Runtime_Total_Minute_CTU_PV,
    CV => Runtime_Total_Minute_CTU_CV); // CTU

// NETWORK 6
Runtime_Total_Hour_CTU(
    CU := Runtime_Total_Minute_CTU.Q,
    RESET := Runtime_Total_Hour_CTU_RESET,
    PV := Runtime_Total_Hour_CTU_PV,
    CV => Runtime_Total); // CTU

// NETWORK 7
Runtime_Maint_Minute_CTU(
    CU := Runtime_TON.Q,
    RESET := Runtime_Maint_Minute_CTU.Q,
    PV := Runtime_Maint_Minute_CTU_PV,
    CV => Runtime_Maint_Minute_CTU_CV); // CTU

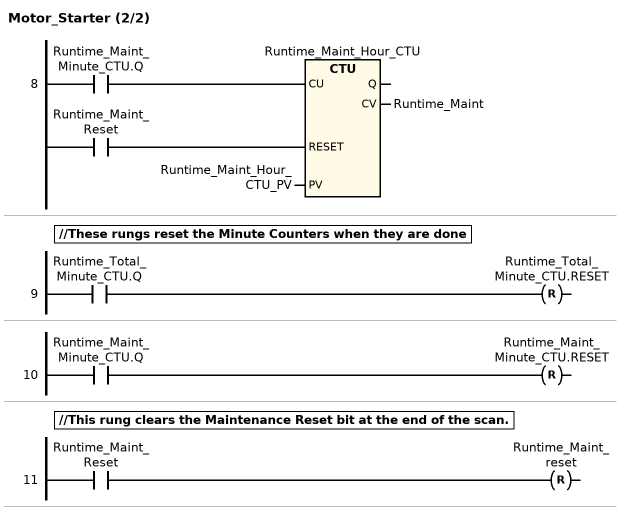
// NETWORK 8
Runtime_Maint_Hour_CTU(
    CU := Runtime_Maint_Minute_CTU.Q,
    RESET := Runtime_Maint_Reset,
    PV := Runtime_Maint_Hour_CTU_PV,
    CV => Runtime_Maint); // CTU

// NETWORK 9
// label: //These rungs reset the Minute Counters when they are done
Runtime_Total_Minute_CTU.RESET R= Runtime_Total_Minute_CTU.Q;

// NETWORK 10
Runtime_Maint_Minute_CTU.RESET R= Runtime_Maint_Minute_CTU.Q;

// NETWORK 11
// label: //This rung clears the Maintenance Reset bit at the end of the scan.
Runtime_Maint_reset R= Runtime_Maint_Reset;

END_FUNCTION_BLOCK

// ---- POUs/Function Blocks/motor_vfd.TcPOU
FUNCTION_BLOCK Motor_VFD
VAR_INPUT
	//Run Feedback from Motor Starter
	Run_Feedback : BOOL; 
	//Reset trigger for Runtime Maint
	Runtime_Maint_Reset : BOOL;
	//Run Request from PLC Program
	Run_Request : BOOL;
	//Requested Speed From PLC Program
	Speed_Request : REAL;
	//Speed Feedback from VFD
	Speed_Feedback : REAL;
	//VFD Fault Status from VFD
	VFD_Fault : BOOL;
	//True if Run Command is true and Run Feedback is false for 3 seconds
	Fail_to_Start : BOOL;
	//True if Run Command is false and Run Feedback is true for 3 seconds
	Fail_to_Stop : BOOL;
	//Daily Reset from GENERAL POU
	Daily_Reset : BOOL;
END_VAR
VAR_OUTPUT
	//Tells the motor to start when true, stop when false
	Run_Command : BOOL;
	//VFD Fault Alarm
	Runtime_Today : REAL;
	//Accumulated Runtime Hours Today
	Runtime_Total : REAL;
	//Resettable Runtime for Maintenance purposes, Description is user adjustable
	Runtime_Maint : REAL;
	//Speed Command to VFD
	Speed_Command : REAL;
END_VAR
VAR
	//Runtime Timer Tags, 1 Minute Timer
	Runtime_TON : TON;
	Runtime_PT : TIME := T#1M;
	Runtime_ET : TIME;
	//Runtime Today Counter
	Runtime_Today_CTU : CTU;
	Runtime_Today_CTU_PV : WORD;
	Runtime_Today_CTU_CV : REAL;
	//Total Runtime Minute Counter
	Runtime_Total_Minute_CTU : CTU;
	Runtime_Total_Minute_CTU_Reset : BOOL;
	Runtime_Total_Minute_CTU_PV : WORD :=60;
	Runtime_Total_Minute_CTU_CV : REAL;
	//Total Runtime Hour Counter
	Runtime_Total_Hour_CTU : CTU;
	Runtime_Total_Hour_CTU_Reset : BOOL;
	Runtime_Total_Hour_CTU_PV : WORD;
	//Maintenance Runtime Minute Counter
	Runtime_Maint_Minute_CTU : CTU;
	Runtime_Maint_Minute_CTU_Reset : BOOL;
	Runtime_Maint_Minute_CTU_PV : WORD :=60;
	Runtime_Maint_Minute_CTU_CV : REAL;
	//Maintenance Runtime Hour Counter
	Runtime_Maint_Hour_CTU : CTU;
	Runtime_Maint_Hour_CTU_PV : WORD;
END_VAR
VAR // added by the converter: edge detectors and wires of the graphical bodies
    _w1, _w2 : BOOL;
END_VAR

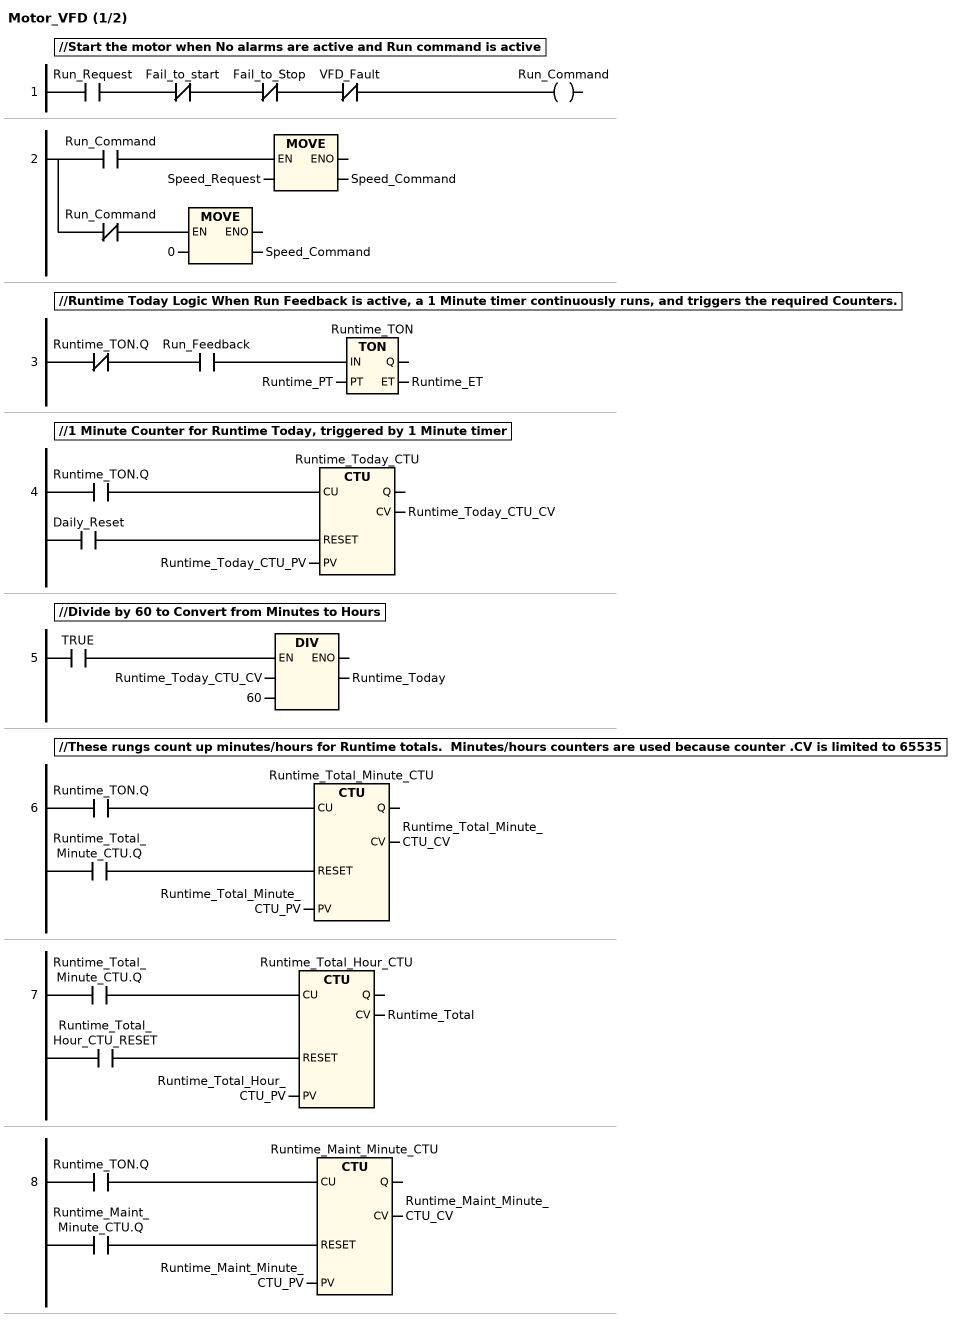
// NETWORK 1
// label: //Start the motor when No alarms are active and Run command is active
Run_Command := Run_Request AND NOT Fail_to_start AND NOT Fail_to_Stop AND NOT VFD_Fault;

// NETWORK 2
_w1 := Run_Command;
IF _w1 THEN Speed_Command := Speed_Request; END_IF
_w2 := NOT Run_Command;
IF _w2 THEN Speed_Command := 0; END_IF
(* _w1 OR _w2; result not used *)

// NETWORK 3
// label: //Runtime Today Logic When Run Feedback is active, a 1 Minute timer continuously runs, and triggers the required Counters.
Runtime_TON(IN := NOT Runtime_TON.Q AND Run_Feedback, PT := Runtime_PT, ET => Runtime_ET); // TON

// NETWORK 4
// label: //1 Minute Counter for Runtime Today, triggered by 1 Minute timer
Runtime_Today_CTU(
    CU := Runtime_TON.Q,
    RESET := Daily_Reset,
    PV := Runtime_Today_CTU_PV,
    CV => Runtime_Today_CTU_CV); // CTU

// NETWORK 5
// label: //Divide by 60 to Convert from Minutes to Hours
Runtime_Today := Runtime_Today_CTU_CV / 60;

// NETWORK 6
// label: //These rungs count up minutes/hours for Runtime totals.  Minutes/hours counters are used because counter .CV is limited to 65535
Runtime_Total_Minute_CTU(
    CU := Runtime_TON.Q,
    RESET := Runtime_Total_Minute_CTU.Q,
    PV := Runtime_Total_Minute_CTU_PV,
    CV => Runtime_Total_Minute_CTU_CV); // CTU

// NETWORK 7
Runtime_Total_Hour_CTU(
    CU := Runtime_Total_Minute_CTU.Q,
    RESET := Runtime_Total_Hour_CTU_RESET,
    PV := Runtime_Total_Hour_CTU_PV,
    CV => Runtime_Total); // CTU

// NETWORK 8
Runtime_Maint_Minute_CTU(
    CU := Runtime_TON.Q,
    RESET := Runtime_Maint_Minute_CTU.Q,
    PV := Runtime_Maint_Minute_CTU_PV,
    CV => Runtime_Maint_Minute_CTU_CV); // CTU

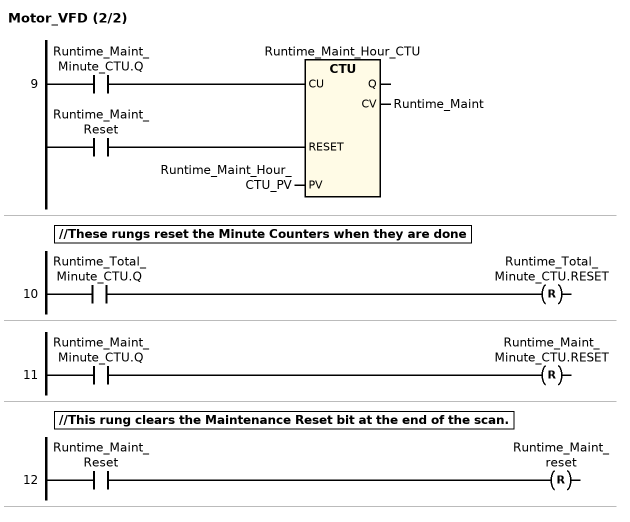
// NETWORK 9
Runtime_Maint_Hour_CTU(
    CU := Runtime_Maint_Minute_CTU.Q,
    RESET := Runtime_Maint_Reset,
    PV := Runtime_Maint_Hour_CTU_PV,
    CV => Runtime_Maint); // CTU

// NETWORK 10
// label: //These rungs reset the Minute Counters when they are done
Runtime_Total_Minute_CTU.RESET R= Runtime_Total_Minute_CTU.Q;

// NETWORK 11
Runtime_Maint_Minute_CTU.RESET R= Runtime_Maint_Minute_CTU.Q;

// NETWORK 12
// label: //This rung clears the Maintenance Reset bit at the end of the scan.
Runtime_Maint_reset R= Runtime_Maint_Reset;

END_FUNCTION_BLOCK

// ---- POUs/Function Blocks/valve_analog.TcPOU
FUNCTION_BLOCK valve_analog
VAR_INPUT
	//Position Feedback from Valve
	position_feedback : REAL; 
	//Position Request from PLC Program
	position_request : REAL;
	//True when valve does not reach position in time
	fault : BOOL;
	// Position deadband for fail to reach position alarm
	position_deadband_sp: REAL;
	//Position valve should move to when faulted
	position_faulted : REAL;
END_VAR
VAR_OUTPUT
	//Position Command to Device
	position_command : REAL;
	// Position Deadband High for fail to reach position alarm
	position_deadband_high: REAL;
	// Position Deadband Low for fail to reach position alarm
	position_deadband_low: REAL;
	// Valve status, 0=Closed, 1=Open, 2=Middle, 3=Faulted
	status: INT;
END_VAR
VAR	
	// Position deadband, calculated value for fail to reach position alarm
	position_deadband: REAL;
	// If position feedback is less than this value, valve status will show closed.
	status_closed_percent: INT :=2;
	// If position feedback is greater than this value, valve status will show open
	status_open_percent : INT :=98;
END_VAR
VAR // added by the converter: edge detectors and wires of the graphical bodies
    _w1, _w2, _w3, _w4, _w5, _w6 : BOOL;
END_VAR

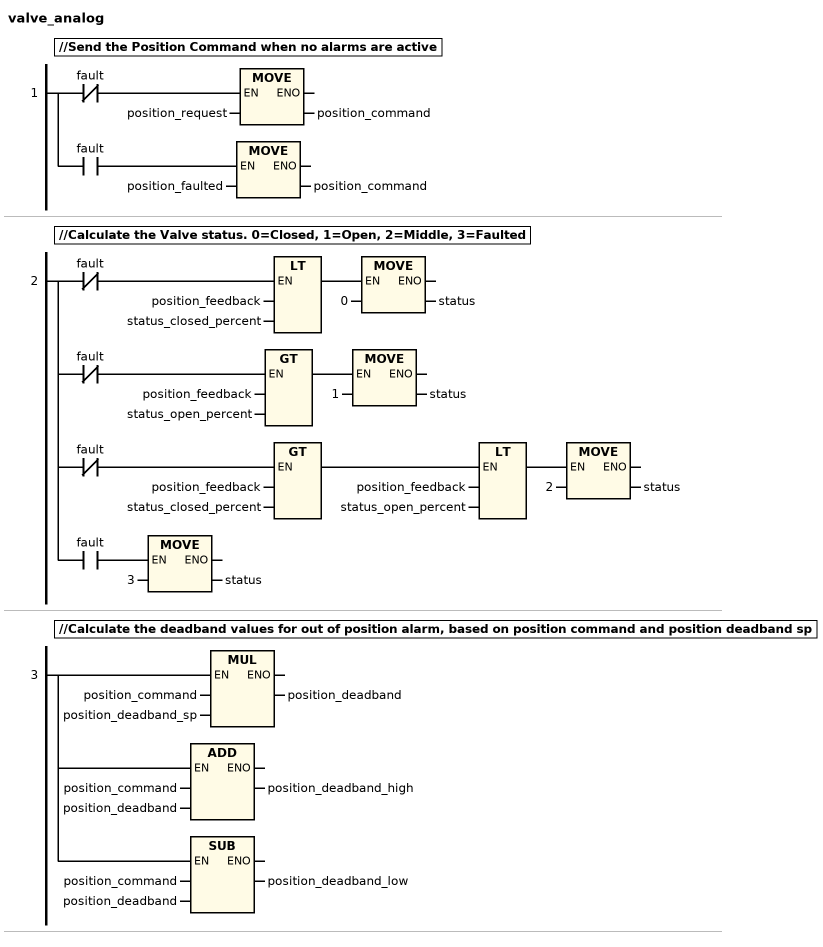
// NETWORK 1
// label: //Send the Position Command when no alarms are active
_w1 := NOT fault;
IF _w1 THEN position_command := position_request; END_IF
_w2 := fault;
IF _w2 THEN position_command := position_faulted; END_IF

// NETWORK 2
// label: //Calculate the Valve status. 0=Closed, 1=Open, 2=Middle, 3=Faulted
_w3 := NOT fault AND position_feedback < status_closed_percent;
IF _w3 THEN status := 0; END_IF
_w4 := NOT fault AND position_feedback > status_open_percent;
IF _w4 THEN status := 1; END_IF
_w5 := NOT fault AND position_feedback > status_closed_percent AND position_feedback < status_open_percent;
IF _w5 THEN status := 2; END_IF
_w6 := fault;
IF _w6 THEN status := 3; END_IF

// NETWORK 3
// label: //Calculate the deadband values for out of position alarm, based on position command and position deadband sp
position_deadband := position_command * position_deadband_sp;
position_deadband_high := position_command + position_deadband;
position_deadband_low := position_command - position_deadband;

END_FUNCTION_BLOCK

// ---- POUs/Function Blocks/valve_digital.TcPOU
FUNCTION_BLOCK valve_digital
VAR_INPUT
	//Open Feedback from Valve
	open_feedback : BOOL; 
	//Closed Feedback from Valve
	closed_feedback : BOOL;
	//Open Request from PLC Program
	open_request : BOOL;
	//Triggered from alarm ladder
	fault : BOOL;
END_VAR
VAR_OUTPUT
	//Tells the valve to open when true, close when False
	open_command : BOOL;
	// Valve status, 0=Closed, 1=Open, 2=Faulted
	status: INT;
END_VAR
VAR	
END_VAR
VAR // added by the converter: edge detectors and wires of the graphical bodies
    _w1, _w2, _w3 : BOOL;
END_VAR

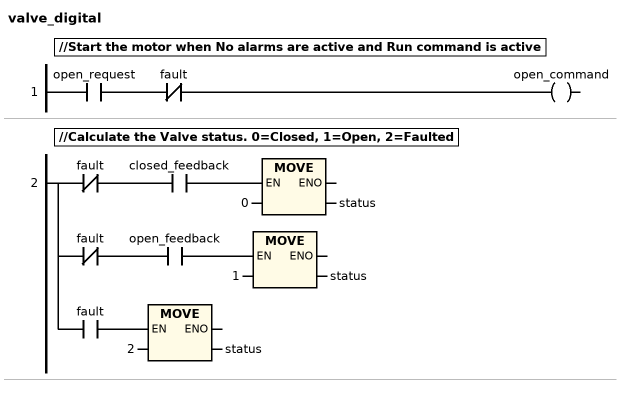
// NETWORK 1
// label: //Start the motor when No alarms are active and Run command is active
open_command := open_request AND NOT fault;

// NETWORK 2
// label: //Calculate the Valve status. 0=Closed, 1=Open, 2=Faulted
_w1 := NOT fault AND closed_feedback;
IF _w1 THEN status := 0; END_IF
_w2 := NOT fault AND open_feedback;
IF _w2 THEN status := 1; END_IF
_w3 := fault;
IF _w3 THEN status := 2; END_IF

END_FUNCTION_BLOCK

// ---- POUs/motor_starter_control_st.TcPOU
PROGRAM motor_starter_control_st
VAR PERSISTENT
	
END_VAR

END_PROGRAM

// ---- POUs/motor_vfd_control_st.TcPOU
PROGRAM motor_vfd_control_st
VAR PERSISTENT
END_VAR

END_PROGRAM

// ---- POUs/valve_analog_control_st.TcPOU
PROGRAM valve_analog_control_st
VAR PERSISTENT

END_VAR

//Instantiate valve analog function block, and map inputs

END_PROGRAM

// ---- POUs/valve_digital_control_st.TcPOU
PROGRAM valve_digital_control_st
VAR PERSISTENT

END_VAR

//Instantiate motor vfd function block, and map inputs

END_PROGRAM
